(*!
<summary>Checks complete STRING/WSTRING ordering beyond the first 255 characters.</summary>
<description>
Builds equal 260-character prefixes followed by different code units. Exercises both operand directions and
both configuration paths, with properly terminated persistent source storage and owned reference snapshots.
Narrow fixture offsets refer to ASCII bytes, including the explicit terminator at offset 261.
</description>
<param name="assertions">Valid assertion context borrowed from the active case.</param>
*)
METHOD PRIVATE testMixedTextComparison
VAR_INPUT
	assertions : REFERENCE TO TOF_Testing.Assertions;
END_VAR
VAR
	i : INT;
END_VAR
_PairComparisonCondition.Comparer := 0;

// SA0175: Build a 260-byte ASCII prefix, one differing byte and a terminator within persistent storage.
{analysis -175}
FOR i := 0 TO 259 DO
	_ComparisonText[i] := BYTE#16#41;
	_ComparisonWideText[i] := WORD#16#41;
END_FOR

_ComparisonText[260] := BYTE#16#42;
_ComparisonWideText[260] := WORD#16#43;
_ComparisonText[261] := TO_BYTE(TOF_Core.UnsignedInt8.MIN_VALUE);
_ComparisonWideText[261] := TO_WORD(TOF_Core.UnsignedInt16.MIN_VALUE);
{analysis +175}

_PairComparisonCondition.BindPlcVariable(name := 'TextNarrow', plcVariable := _ComparisonText);
_PairComparisonCondition.BindPlcVariable(name := 'TextWide', plcVariable := _ComparisonWideText);

_PairComparisonCondition.ConfigureVariable(
	firstVariableName := 'TextNarrow',
	comparisonOperator := TOF_Workflow.COMPARISON_OPERATOR.LESS_THAN,
	secondVariableName := 'TextWide'
);
assertions.ThatBool(
	actual := _PairComparisonCondition.Evaluate(activity := 0),
	message := "Mixed text must compare beyond character 255"
).IsTrue();

_PairComparisonCondition.ConfigureVariable(
	firstVariableName := 'TextWide',
	comparisonOperator := TOF_Workflow.COMPARISON_OPERATOR.GREATER_THAN,
	secondVariableName := 'TextNarrow'
);
assertions.ThatBool(
	actual := _PairComparisonCondition.Evaluate(activity := 0),
	message := "Reversing mixed encodings must reverse order"
).IsTrue();

_PairComparisonCondition.Configure(
	firstVariableName := 'TextNarrow',
	comparisonOperator := TOF_Workflow.COMPARISON_OPERATOR.LESS_THAN,
	referenceValue := _ComparisonWideText
);
assertions.ThatBool(
	actual := _PairComparisonCondition.Evaluate(activity := 0),
	message := "A long WSTRING reference must compare fully"
).IsTrue();

_PairComparisonCondition.Configure(
	firstVariableName := 'TextWide',
	comparisonOperator := TOF_Workflow.COMPARISON_OPERATOR.GREATER_THAN,
	referenceValue := _ComparisonText
);
assertions.ThatBool(
	actual := _PairComparisonCondition.Evaluate(activity := 0),
	message := "A long STRING reference must compare fully"
).IsTrue();
END_METHOD

(*!
<summary>Checks that equal-category time-of-day and user-defined pairs retain standard comparer dispatch.</summary>
<description>
Uses categories unsupported by built-in GENERIC_VALUE.CompareTo. Time-of-day values retain native order and
user-defined unions retain explicit byte order, including when a reference snapshot is configured.
</description>
<param name="assertions">Valid assertion context borrowed from the active case.</param>
*)
METHOD PRIVATE testStandardComparisonFallback
VAR_INPUT
	assertions : REFERENCE TO TOF_Testing.Assertions;
END_VAR
_PairComparisonCondition.Comparer := 0;
_FirstComparisonBytes.Raw := UDINT#16#01010101;
_SecondComparisonBytes.Raw := UDINT#16#02020202;

_PairComparisonCondition.BindPlcVariable(name := 'FallbackEarlierTime', plcVariable := _FirstComparisonTimeOfDay);
_PairComparisonCondition.BindPlcVariable(name := 'FallbackLaterTime', plcVariable := _SecondComparisonTimeOfDay);
_PairComparisonCondition.BindPlcVariable(name := 'FallbackFirstBytes', plcVariable := _FirstComparisonBytes);
_PairComparisonCondition.BindPlcVariable(name := 'FallbackSecondBytes', plcVariable := _SecondComparisonBytes);

_PairComparisonCondition.ConfigureVariable(
	firstVariableName := 'FallbackEarlierTime',
	comparisonOperator := TOF_Workflow.COMPARISON_OPERATOR.LESS_THAN,
	secondVariableName := 'FallbackLaterTime'
);
assertions.ThatBool(
	actual := _PairComparisonCondition.Evaluate(activity := 0),
	message := "TIME_OF_DAY must retain native ordering"
).IsTrue();

_PairComparisonCondition.Configure(
	firstVariableName := 'FallbackLaterTime',
	comparisonOperator := TOF_Workflow.COMPARISON_OPERATOR.GREATER_THAN,
	referenceValue := _FirstComparisonTimeOfDay
);
assertions.ThatBool(
	actual := _PairComparisonCondition.Evaluate(activity := 0),
	message := "A time-of-day reference must remain supported"
).IsTrue();

_PairComparisonCondition.ConfigureVariable(
	firstVariableName := 'FallbackFirstBytes',
	comparisonOperator := TOF_Workflow.COMPARISON_OPERATOR.LESS_THAN,
	secondVariableName := 'FallbackSecondBytes'
);
assertions.ThatBool(
	actual := _PairComparisonCondition.Evaluate(activity := 0),
	message := "USER_DEFINED must retain byte ordering"
).IsTrue();

_PairComparisonCondition.Configure(
	firstVariableName := 'FallbackSecondBytes',
	comparisonOperator := TOF_Workflow.COMPARISON_OPERATOR.GREATER_THAN,
	referenceValue := _FirstComparisonBytes
);
assertions.ThatBool(
	actual := _PairComparisonCondition.Evaluate(activity := 0),
	message := "A user-defined reference must remain supported"
).IsTrue();
END_METHOD

(*!
<summary>Checks rejection of unrelated categories before standard typed payload comparison.</summary>
<description>
Exercises equal-width numeric/time pairs, numeric/text pairs and OBJECT/USER_DEFINED in both directions.
Both configuration paths are evaluated. Expected exceptions are checked by interface category; a valid
comparison afterwards verifies that failed evaluation preserves reusable configuration state.
</description>
<param name="assertions">Valid assertion context borrowed from the active case.</param>
*)
METHOD PRIVATE testIncompatibleComparisonPairs
VAR_INPUT
	assertions : REFERENCE TO TOF_Testing.Assertions;
END_VAR
_PairComparisonCondition.Comparer := 0;
_PairComparisonCondition.BindPlcVariable(name := 'RejectedNumber', plcVariable := _ComparisonUnrelatedInteger);
_PairComparisonCondition.BindPlcVariable(name := 'RejectedTime', plcVariable := _FirstComparisonTimeOfDay);
_PairComparisonCondition.BindPlcVariable(name := 'RejectedText', plcVariable := _ComparisonText);
_PairComparisonCondition.BindPlcVariable(name := 'RejectedBytes', plcVariable := _FirstComparisonBytes);
_PairComparisonCondition.BindPlcVariable(
	name := 'RejectedObject',
	plcVariable := _ComparisonObject,
	plcVariableIsObject := TRUE
);

_PairComparisonCondition.ConfigureVariable(
	firstVariableName := 'RejectedNumber',
	comparisonOperator := TOF_Workflow.COMPARISON_OPERATOR.EQUAL,
	secondVariableName := 'RejectedTime'
);
assertComparisonRejected(
	assertions := assertions,
	scenario := 'DINT/TOD variables');

_PairComparisonCondition.ConfigureVariable(
	firstVariableName := 'RejectedTime',
	comparisonOperator := TOF_Workflow.COMPARISON_OPERATOR.EQUAL,
	secondVariableName := 'RejectedNumber'
);
assertComparisonRejected(
	assertions := assertions,
	scenario := 'TOD/DINT variables');

_PairComparisonCondition.Configure(
	firstVariableName := 'RejectedNumber',
	comparisonOperator := TOF_Workflow.COMPARISON_OPERATOR.EQUAL,
	referenceValue := _FirstComparisonTimeOfDay
);
assertComparisonRejected(
	assertions := assertions,
	scenario := 'DINT/TOD reference');

_PairComparisonCondition.Configure(
	firstVariableName := 'RejectedTime',
	comparisonOperator := TOF_Workflow.COMPARISON_OPERATOR.EQUAL,
	referenceValue := _ComparisonUnrelatedInteger
);
assertComparisonRejected(
	assertions := assertions,
	scenario := 'TOD/DINT reference');

_PairComparisonCondition.ConfigureVariable(
	firstVariableName := 'RejectedNumber',
	comparisonOperator := TOF_Workflow.COMPARISON_OPERATOR.EQUAL,
	secondVariableName := 'RejectedText'
);
assertComparisonRejected(
	assertions := assertions,
	scenario := 'DINT/STRING variables');

_PairComparisonCondition.ConfigureVariable(
	firstVariableName := 'RejectedText',
	comparisonOperator := TOF_Workflow.COMPARISON_OPERATOR.EQUAL,
	secondVariableName := 'RejectedNumber'
);
assertComparisonRejected(
	assertions := assertions,
	scenario := 'STRING/DINT variables');

_PairComparisonCondition.ConfigureVariable(
	firstVariableName := 'RejectedObject',
	comparisonOperator := TOF_Workflow.COMPARISON_OPERATOR.EQUAL,
	secondVariableName := 'RejectedBytes'
);
assertComparisonRejected(
	assertions := assertions,
	scenario := 'OBJECT/USER_DEFINED variables');

_PairComparisonCondition.ConfigureVariable(
	firstVariableName := 'RejectedBytes',
	comparisonOperator := TOF_Workflow.COMPARISON_OPERATOR.EQUAL,
	secondVariableName := 'RejectedObject'
);
assertComparisonRejected(
	assertions := assertions,
	scenario := 'USER_DEFINED/OBJECT variables');

_PairComparisonCondition.Configure(
	firstVariableName := 'RejectedNumber',
	comparisonOperator := TOF_Workflow.COMPARISON_OPERATOR.EQUAL,
	referenceValue := _ComparisonUnrelatedInteger
);
assertions.ThatBool(
	actual := _PairComparisonCondition.Evaluate(activity := 0),
	message := "The condition must remain usable after rejection"
).IsTrue();
END_METHOD

(*!
<summary>Evaluates the configured pair and asserts the expected unsupported-conversion exception category.</summary>
<description>
Converts an expected configuration failure into a test diagnostic. Unexpected exception categories fail the
assertion. Captured exception interfaces remain borrowed within this call and are not retained after task
cleanup. The persistent condition owns all resources across the exception boundary.
</description>
<param name="scenario">Short label identifying the rejected operand pair in assertion diagnostics.</param>
<param name="assertions">Valid assertion context borrowed from the active case.</param>
*)
METHOD PRIVATE assertComparisonRejected
VAR_INPUT
	assertions : REFERENCE TO TOF_Testing.Assertions;
	scenario : STRING(255);
END_VAR
VAR
	exceptionCode : __SYSTEM.ExceptionCode;
	caughtException : TOF_Core.IException;
	conversionException : TOF_Core.IGenericConversionNotSupportedException;
	caughtExpectedException : BOOL;
END_VAR
__TRY
	_PairComparisonCondition.Evaluate(activity := 0);
__CATCH(exceptionCode)
	caughtException := TOF_Core.ExceptionManager.GetLastException(
		exceptionCode := exceptionCode,
		catchPointNamespaceName := NamespaceName,
		catchPointPOUName := __POUNAME(),
		catchPointPosition := __POSITION()
	);
	caughtExpectedException := __QUERYINTERFACE(caughtException, conversionException);
__ENDTRY

assertions.ThatBool(
	actual := caughtExpectedException,
	message := TO_WSTRING(TOF_Core.Strings.Concat255(scenario, ': expected GenericConversionNotSupportedException'))
).IsTrue();
assertions.ThatBool(
	actual := _PairComparisonCondition.Configured,
	message := TO_WSTRING(TOF_Core.Strings.Concat255(scenario, ': rejected evaluation must preserve configuration'))
).IsTrue();
END_METHOD

(*!
<summary>Runs the packaging and inspection workflow through completion and exception recovery.</summary>
<param name="assertions">Valid assertion context borrowed from the active case.</param>
*)
METHOD PRIVATE testEndToEndComprehensiveScenario
VAR_INPUT
	assertions : REFERENCE TO TOF_Testing.Assertions;
END_VAR
VAR
	cycleIndex : INT;
END_VAR
buildScenarioTree();

_Workflow.SensorFeedPart := FALSE; // will be set TRUE by parallelStep
_Workflow.SensorVacuumOk := TRUE;
_Workflow.SensorInspectionOk := TRUE;

assertions.ThatBool(
	actual := _Workflow.StartingAllowed,
	message := "Workflow must allow starting from PASSIVE_READY"
).IsTrue();
_Workflow.RequestStart();

FOR cycleIndex := 1 TO 200 DO
	_Workflow.Execute();

	IF NOT _Workflow.Busy THEN
		EXIT;
	END_IF
END_FOR

assertions.ThatBool(
	actual := _Workflow.State = TOF_Workflow.WORKFLOW_ELEMENT_STATE.PASSIVE_COMPLETED,
	message := "Workflow must complete with PASSIVE_COMPLETED"
).IsTrue();
assertions.ThatInt(
	actual := _Workflow.ProducedCount,
	message := "ProducedCount must equal 1 after WhileActivity and AssignVariableActivity"
).ToBe(expected := 1);
assertions.ThatBool(
	actual := _Workflow.ErrorHandled,
	message := "ErrorHandled must be TRUE after CatchActivity recovered from Try exception"
).IsTrue();
assertions.ThatBool(
	actual := _ThrowingActivity.ThrowCount > 0,
	message := "ThrowingActivity must have executed and thrown"
).IsTrue();
END_METHOD

(*!
<summary>Checks NotCondition using persistent resource-owning fixtures.</summary>
<description>Fixture allocations remain owned by the suite across unexpected exception propagation.</description>
<param name="assertions">Valid assertion context borrowed from the active case.</param>
*)
METHOD PRIVATE testNotCondition
VAR_INPUT
	assertions : REFERENCE TO TOF_Testing.Assertions;
END_VAR
VAR_INST
	notCond : TOF_Workflow.NotCondition(workflow := _NotWorkflow);
	trueCond : TOF_Workflow.TrueCondition(workflow := _NotWorkflow);
	varCond : TOF_Workflow.VariableHasValueCondition(workflow := _NotWorkflow);
	testVal : INT := 10;
END_VAR
_NotWorkflow.SetRootActivity(rootActivity := _NotRoot);

assertions.ThatBool(
	actual := notCond.Configured,
	message := "NotCondition must not be configured initially"
).IsFalse();

notCond.Configure(condition := trueCond);
assertions.ThatBool(
	actual := notCond.Configured,
	message := "NotCondition must be configured after Configure"
).IsTrue();
assertions.ThatBool(
	actual := notCond.Evaluate(activity := 0),
	message := "NOT True must evaluate to FALSE"
).IsFalse();

_NotWorkflow.ProducedCount := testVal;
varCond.Configure(monitoredVariableName := 'ProducedCount', referenceValue := testVal);
notCond.Configure(condition := varCond);
assertions.ThatBool(
	actual := notCond.Evaluate(activity := 0),
	message := "NOT (ProducedCount = 10) when ProducedCount = 10 must be FALSE"
).IsFalse();

_NotWorkflow.ProducedCount := 99;
assertions.ThatBool(
	actual := notCond.Evaluate(activity := 0),
	message := "NOT (ProducedCount = 10) when ProducedCount = 99 must be TRUE"
).IsTrue();
END_METHOD

(*!
<summary>Checks ParallelActivityWaitAll using persistent resource-owning fixtures.</summary>
<description>Fixture allocations remain owned by the suite across unexpected exception propagation.</description>
<param name="assertions">Valid assertion context borrowed from the active case.</param>
*)
METHOD PRIVATE testParallelActivityWaitAll
VAR_INPUT
	assertions : REFERENCE TO TOF_Testing.Assertions;
END_VAR
VAR_INST
	parallelAct : TOF_Workflow.ParallelActivity(workflow := _WaitAllWorkflow);
	counterTask1 : CounterTask(name := "WaitAllCounter1");
	counterTask2 : CounterTask(name := "WaitAllCounter2");
	taskAct1 : TOF_Workflow.InvokeTaskActivity(workflow := _WaitAllWorkflow);
	taskAct2 : TOF_Workflow.InvokeTaskActivity(workflow := _WaitAllWorkflow);
	cycleIndex : INT;
	refuseReason : TOF_Core.ERROR_MESSAGE;
END_VAR
counterTask1.Reset(refuseReason => refuseReason);
counterTask1.TargetValue := 1;
taskAct1.Configure(task := counterTask1);

counterTask2.Reset(refuseReason => refuseReason);
counterTask2.TargetValue := 2;
taskAct2.Configure(task := counterTask2);

parallelAct.Mode := TOF_Workflow.PARALLEL_JOIN_MODE.WAIT_ALL;
parallelAct.AddChildActivity(activity := taskAct1);
parallelAct.AddChildActivity(activity := taskAct2);

assertions.ThatDInt(actual := parallelAct.ChildCount, message := "ChildCount must be 2").ToBe(expected := 2);

parallelAct.RequestStart();
assertions.ThatBool(
	actual := parallelAct.Busy,
	message := "ParallelActivity must be busy after RequestStart"
).IsTrue();

FOR cycleIndex := 1 TO 50 DO
	parallelAct.Execute();

	IF NOT parallelAct.Busy THEN
		EXIT;
	END_IF
END_FOR

	assertions.ThatBool(
		actual := parallelAct.State = TOF_Workflow.WORKFLOW_ELEMENT_STATE.PASSIVE_COMPLETED,
		message := "ParallelActivity with WAIT_ALL must complete with PASSIVE_COMPLETED"
	).IsTrue();
assertions.ThatBool(
	actual := taskAct1.State = TOF_Workflow.WORKFLOW_ELEMENT_STATE.PASSIVE_COMPLETED,
	message := "taskAct1 must be PASSIVE_COMPLETED"
).IsTrue();
assertions.ThatBool(
	actual := taskAct2.State = TOF_Workflow.WORKFLOW_ELEMENT_STATE.PASSIVE_COMPLETED,
	message := "taskAct2 must be PASSIVE_COMPLETED"
).IsTrue();

parallelAct.RequestReset();
assertions.ThatBool(
	actual := parallelAct.State = TOF_Workflow.WORKFLOW_ELEMENT_STATE.PASSIVE_READY,
	message := "ParallelActivity must reset to PASSIVE_READY"
).IsTrue();
assertions.ThatBool(
	actual := taskAct1.State = TOF_Workflow.WORKFLOW_ELEMENT_STATE.PASSIVE_READY,
	message := "taskAct1 must reset to PASSIVE_READY"
).IsTrue();
assertions.ThatBool(
	actual := taskAct2.State = TOF_Workflow.WORKFLOW_ELEMENT_STATE.PASSIVE_READY,
	message := "taskAct2 must reset to PASSIVE_READY"
).IsTrue();
END_METHOD

(*!
<summary>Checks ParallelActivityWaitAny using persistent resource-owning fixtures.</summary>
<description>Fixture allocations remain owned by the suite across unexpected exception propagation.</description>
<param name="assertions">Valid assertion context borrowed from the active case.</param>
*)
METHOD PRIVATE testParallelActivityWaitAny
VAR_INPUT
	assertions : REFERENCE TO TOF_Testing.Assertions;
END_VAR
VAR_INST
	parallelAct : TOF_Workflow.ParallelActivity(workflow := _WaitAnyWorkflow);
	fastAssign : TOF_Workflow.AssignVariableActivity(workflow := _WaitAnyWorkflow);
	longDelay : TOF_Workflow.DelayActivity(workflow := _WaitAnyWorkflow);
	cycleIndex : INT;
	val : INT := 42;
END_VAR
_WaitAnyWorkflow.SetRootActivity(rootActivity := _WaitAnyRoot);

fastAssign.Configure(targetVariableName := 'ProducedCount', value := val);
longDelay.Interval := T#10S;

parallelAct.Mode := TOF_Workflow.PARALLEL_JOIN_MODE.WAIT_ANY;
parallelAct.AddChildActivity(activity := fastAssign);
parallelAct.AddChildActivity(activity := longDelay);

parallelAct.RequestStart();

FOR cycleIndex := 1 TO 20 DO
	parallelAct.Execute();

	IF NOT parallelAct.Busy THEN
		EXIT;
	END_IF
END_FOR

	assertions.ThatBool(
		actual := parallelAct.State = TOF_Workflow.WORKFLOW_ELEMENT_STATE.PASSIVE_COMPLETED,
		message := "ParallelActivity with WAIT_ANY must complete once fast branch finishes"
	).IsTrue();
assertions.ThatBool(
	actual := fastAssign.State = TOF_Workflow.WORKFLOW_ELEMENT_STATE.PASSIVE_COMPLETED,
	message := "fastAssign must be PASSIVE_COMPLETED"
).IsTrue();
	assertions.ThatBool(
		actual := longDelay.State = TOF_Workflow.WORKFLOW_ELEMENT_STATE.PASSIVE_CANCELLED,
		message := "longDelay must be cancelled when sibling branch completed under WAIT_ANY"
	).IsTrue();

parallelAct.RequestReset();
assertions.ThatBool(
	actual := parallelAct.State = TOF_Workflow.WORKFLOW_ELEMENT_STATE.PASSIVE_READY,
	message := "ParallelActivity must reset to PASSIVE_READY"
).IsTrue();
END_METHOD

(*!
<summary>Checks that a started workflow accepts cancellation and reaches its cancelled state.</summary>
<param name="assertions">Valid assertion context borrowed from the active case.</param>
*)
METHOD PRIVATE testWorkflowCancel
VAR_INPUT
	assertions : REFERENCE TO TOF_Testing.Assertions;
END_VAR
VAR
	cycleIndex : INT;
END_VAR
buildScenarioTree();

_Workflow.SensorVacuumOk := FALSE; // keep waiting at condition
_Workflow.RequestStart();

assertions.ThatBool(
	actual := _Workflow.CancellingAllowed,
	message := "Workflow must allow cancelling while busy"
).IsTrue();
_Workflow.RequestCancel(reason := "Cancelled by test");

FOR cycleIndex := 1 TO 20 DO
	_Workflow.Execute();

	IF NOT _Workflow.Busy THEN
		EXIT;
	END_IF
END_FOR

assertions.ThatBool(
	actual := _Workflow.State = TOF_Workflow.WORKFLOW_ELEMENT_STATE.PASSIVE_CANCELLED,
	message := "Workflow must transition to PASSIVE_CANCELLED"
).IsTrue();
END_METHOD

(*!
<summary>Checks WorkflowReset with an independently prepared workflow fixture.</summary>
<description>
Assertions run unconditionally after preparing the required state; other test outcomes are not prerequisites.
</description>
<param name="assertions">Valid assertion context borrowed from the active case.</param>
*)
METHOD PRIVATE testWorkflowReset
VAR_INPUT
	assertions : REFERENCE TO TOF_Testing.Assertions;
END_VAR
VAR
	cycleIndex : INT;
END_VAR
_ResetActivity.Interval := T#0S;
_ResetWorkflow.SetRootActivity(rootActivity := _ResetActivity);
_ResetWorkflow.ProducedCount := 7;
_ResetWorkflow.ErrorHandled := TRUE;
_ResetWorkflow.RequestStart();

FOR cycleIndex := 1 TO 20 DO
	_ResetWorkflow.Execute();

	IF NOT _ResetWorkflow.Busy THEN
		EXIT;
	END_IF
END_FOR

assertions.ThatBool(
	actual := _ResetWorkflow.State = TOF_Workflow.WORKFLOW_ELEMENT_STATE.PASSIVE_COMPLETED,
	message := "The independent reset fixture must finish its run"
).IsTrue();
assertions.ThatBool(
	actual := _ResetWorkflow.ResettingAllowed,
	message := "A completed workflow must allow reset"
).IsTrue();
_ResetWorkflow.RequestReset();

FOR cycleIndex := 1 TO 20 DO
	_ResetWorkflow.Execute();

	IF NOT _ResetWorkflow.Busy THEN
		EXIT;
	END_IF
END_FOR

assertions.ThatBool(
	actual := _ResetWorkflow.State = TOF_Workflow.WORKFLOW_ELEMENT_STATE.PASSIVE_READY,
	message := "Reset must restore PASSIVE_READY"
).IsTrue();
assertions.ThatInt(
	actual := _ResetWorkflow.ProducedCount,
	message := "Reset must clear ProducedCount"
).ToBe(expected := 0);
assertions.ThatBool(actual := _ResetWorkflow.ErrorHandled, message := "Reset must clear ErrorHandled").IsFalse();
END_METHOD

(*!
<summary>Checks concrete dynamic Workflow creation, variable binding and deletion.</summary>
<description>The suite tracks the pointer persistently until explicit deletion or suite destruction.</description>
<param name="assertions">Valid assertion context borrowed from the active case.</param>
*)
METHOD PRIVATE testDirectWorkflowDynamicCreation
VAR_INPUT
	assertions : REFERENCE TO TOF_Testing.Assertions;
END_VAR
VAR
	resolvedVar : TOF_Core.GENERIC_VALUE;
	registered : BOOL;
	found : BOOL;
END_VAR
_DirectWorkflow := __NEW(TOF_Workflow.Workflow);

IF _DirectWorkflow = 0 THEN
	TOF_Core.DynamicMemoryManager.RaiseAllocationFailure();
END_IF

assertions.ThatBool(
	actual := _DirectWorkflow <> 0,
	message := "Workflow dynamic creation (__NEW) must succeed"
).IsTrue();

IF _DirectWorkflow <> 0 THEN
	registered := _DirectWorkflow^.BindPlcVariable(name := 'DynamicVar', plcVariable := _DynamicTestVar);
	assertions.ThatBool(
		actual := registered,
		message := "BindPlcVariable on dynamic Workflow must return TRUE"
	).IsTrue();

	found := _DirectWorkflow^.TryGetVariable(name := 'DynamicVar', variable => resolvedVar);
	assertions.ThatBool(
		actual := found,
		message := "TryGetVariable on dynamic Workflow must find registered variable"
	).IsTrue();
	assertions.ThatBool(
		actual := resolvedVar.Address = ADR(_DynamicTestVar),
		message := "Resolved variable address must match"
	).IsTrue();

	__DELETE(_DirectWorkflow);
	assertions.ThatBool(
		actual := _DirectWorkflow = 0,
		message := "Workflow dynamic deletion (__DELETE) must succeed"
	).IsTrue();
END_IF
END_METHOD

(*!
<summary>Checks ActivityVariableScopingAndShadowing with an independently prepared workflow fixture.</summary>
<description>
Assertions run unconditionally after preparing the required state; other test outcomes are not prerequisites.
</description>
<param name="assertions">Valid assertion context borrowed from the active case.</param>
*)
METHOD PRIVATE testActivityVariableScopingAndShadowing
VAR_INPUT
	assertions : REFERENCE TO TOF_Testing.Assertions;
END_VAR
VAR
	rootSequence : POINTER TO TOF_Workflow.SequenceActivity;
	childAssign : POINTER TO TOF_Workflow.AssignVariableActivity;
	resolvedVar : TOF_Core.GENERIC_VALUE;
	found : BOOL;
END_VAR
rootSequence := __NEW(TOF_Workflow.SequenceActivity(workflow := _ScopeWorkflow));

IF rootSequence = 0 THEN
	TOF_Core.DynamicMemoryManager.RaiseAllocationFailure();
END_IF

_Workflow.RegisterChild(child := rootSequence^);

childAssign := __NEW(TOF_Workflow.AssignVariableActivity(workflow := _ScopeWorkflow));

IF childAssign = 0 THEN
	TOF_Core.DynamicMemoryManager.RaiseAllocationFailure();
END_IF

_Workflow.RegisterChild(child := childAssign^);

rootSequence^.AddChildActivity(activity := childAssign^);

// Register variable in parent activity scope
rootSequence^.BindPlcVariable(name := 'ParentVar', plcVariable := _ParentScopeVar);

// Child should find parent variable through hierarchical resolution
found := childAssign^.TryGetVariable(name := 'ParentVar', variable => resolvedVar);
assertions.ThatBool(
	actual := found,
	message := "Child activity must resolve variable from parent activity scope"
).IsTrue();
assertions.ThatBool(
	actual := resolvedVar.Address = ADR(_ParentScopeVar),
	message := "Parent variable address must match"
).IsTrue();

// Register variable in workflow, and shadow it in child activity
_ScopeWorkflow.BindPlcVariable(name := 'ShadowVar', plcVariable := _WorkflowScopeVar);
childAssign^.BindPlcVariable(name := 'ShadowVar', plcVariable := _ChildLocalVar);

// Child activity must resolve its own shadowed local variable
found := childAssign^.TryGetVariable(name := 'ShadowVar', variable => resolvedVar);
assertions.ThatBool(actual := found, message := "Child activity must resolve its own shadowed variable").IsTrue();
assertions.ThatBool(
	actual := resolvedVar.Address = ADR(_ChildLocalVar),
	message := "Shadowed variable must point to child local address"
).IsTrue();

// Workflow must resolve its own global variable
found := _ScopeWorkflow.TryGetVariable(name := 'ShadowVar', variable => resolvedVar);
assertions.ThatBool(actual := found, message := "Workflow must resolve its own variable").IsTrue();
assertions.ThatBool(
	actual := resolvedVar.Address = ADR(_WorkflowScopeVar),
	message := "Workflow variable must point to workflow address"
).IsTrue();
END_METHOD

(*!
<summary>Checks VariableRegistrationValidation with an independently prepared workflow fixture.</summary>
<description>
Assertions run unconditionally after preparing the required state; other test outcomes are not prerequisites.
</description>
<param name="assertions">Valid assertion context borrowed from the active case.</param>
*)
METHOD PRIVATE testVariableRegistrationValidation
VAR_INPUT
	assertions : REFERENCE TO TOF_Testing.Assertions;
END_VAR
VAR
	stackValue : INT;
	exceptionCode : __SYSTEM.ExceptionCode;
	exception : TOF_Core.IException;
	configurationException : TOF_Workflow.IWorkflowConfigurationException;
	caughtExpected : BOOL;
END_VAR
_ValidationWorkflow.BindPlcVariable(name := 'Registered', plcVariable := _ValidationValue);

__TRY
	_ValidationWorkflow.BindPlcVariable(name := 'StackValue', plcVariable := stackValue);
__CATCH(exceptionCode)
	exception := TOF_Core.ExceptionManager.GetLastException(
		exceptionCode := exceptionCode,
		catchPointNamespaceName := NamespaceName,
		catchPointPOUName := __POUNAME(),
		catchPointPosition := __POSITION()
	);
	caughtExpected := __QUERYINTERFACE(exception, configurationException);
__ENDTRY

assertions.ThatBool(
	actual := caughtExpected,
	message := "Stack binding must raise WorkflowConfigurationException"
).IsTrue();
caughtExpected := FALSE;

__TRY
	_ValidationWorkflow.BindPlcVariable(name := '', plcVariable := _ValidationValue);
__CATCH(exceptionCode)
	exception := TOF_Core.ExceptionManager.GetLastException(
		exceptionCode := exceptionCode,
		catchPointNamespaceName := NamespaceName,
		catchPointPOUName := __POUNAME(),
		catchPointPosition := __POSITION()
	);
	caughtExpected := __QUERYINTERFACE(exception, configurationException);
__ENDTRY

assertions.ThatBool(
	actual := caughtExpected,
	message := "Empty name must raise WorkflowConfigurationException"
).IsTrue();
caughtExpected := FALSE;

__TRY
	_ValidationWorkflow.BindPlcVariable(name := 'Registered', plcVariable := _ValidationValue);
__CATCH(exceptionCode)
	exception := TOF_Core.ExceptionManager.GetLastException(
		exceptionCode := exceptionCode,
		catchPointNamespaceName := NamespaceName,
		catchPointPOUName := __POUNAME(),
		catchPointPosition := __POSITION()
	);
	caughtExpected := __QUERYINTERFACE(exception, configurationException);
__ENDTRY

assertions.ThatBool(
	actual := caughtExpected,
	message := "Duplicate persistent binding must raise configuration failure"
).IsTrue();

_ValidationActivity.Interval := T#10S;
_ValidationWorkflow.SetRootActivity(rootActivity := _ValidationActivity);
_ValidationWorkflow.RequestStart();
assertions.ThatBool(
	actual := _ValidationWorkflow.Busy,
	message := "The busy guard fixture must actually be active"
).IsTrue();
caughtExpected := FALSE;

__TRY
	_ValidationWorkflow.BindPlcVariable(name := 'WhileBusy', plcVariable := _ValidationValue);
__CATCH(exceptionCode)
	exception := TOF_Core.ExceptionManager.GetLastException(
		exceptionCode := exceptionCode,
		catchPointNamespaceName := NamespaceName,
		catchPointPOUName := __POUNAME(),
		catchPointPosition := __POSITION()
	);
	caughtExpected := __QUERYINTERFACE(exception, configurationException);
__ENDTRY

_ValidationWorkflow.RequestCancel(reason := "Validation complete");
_ValidationWorkflow.RequestReset();
assertions.ThatBool(
	actual := caughtExpected,
	message := "Busy registration must raise configuration failure"
).IsTrue();
END_METHOD

(*!
<summary>Releases any direct-creation fixture still owned by the suite.</summary>
<description>
Completes without exceptions; registered scenario nodes remain owned by their workflow fields.
</description>
*)
METHOD FB_exit : BOOL
VAR_INPUT
	bInCopyCode : BOOL;
END_VAR
IF NOT bInCopyCode AND_THEN _DirectWorkflow <> 0 THEN
	__DELETE(_DirectWorkflow);
END_IF
END_METHOD

END_FUNCTION_BLOCK

// ---- Tests/Workflow/ComprehensiveTestWorkflow.TcPOU
(*
SPDX-FileCopyrightText: © 2026 Oleksandr Tiutyk <trofimich@gmail.com>
SPDX-License-Identifier: MIT
License: https://opensource.org/license/mit
*)

(*!
<summary>Test workflow instance containing named variables for the comprehensive workflow scenario test.</summary>
*)

{attribute 'no_explicit_call' := 'do not call this function block directly'}
{attribute 'enable_dynamic_creation'}
FUNCTION_BLOCK ComprehensiveTestWorkflow EXTENDS TOF_Workflow.Workflow
VAR_INPUT
	SensorFeedPart : BOOL;
	SensorVacuumOk : BOOL;
	SensorInspectionOk : BOOL;
	BatchTarget : INT;
	ProducedCount : INT;
	RejectCount : INT;
	ErrorHandled : BOOL;
END_VAR
VAR_STAT
	//! <summary>Concrete test workflow name available during inherited initialization.</summary>
	_TestWorkflowClassName : STRING := __POUNAME();
END_VAR

METHOD PROTECTED InitializeVariables
BindPlcVariable(name := 'BatchTarget', plcVariable := BatchTarget);
BindPlcVariable(name := 'ProducedCount', plcVariable := ProducedCount);
BindPlcVariable(name := 'RejectCount', plcVariable := RejectCount);
BindPlcVariable(name := 'SensorFeedPart', plcVariable := SensorFeedPart);
BindPlcVariable(name := 'SensorVacuumOk', plcVariable := SensorVacuumOk);
BindPlcVariable(name := 'SensorInspectionOk', plcVariable := SensorInspectionOk);
BindPlcVariable(name := 'ErrorHandled', plcVariable := ErrorHandled);
END_METHOD

{attribute 'monitoring' := 'call'}
PROPERTY NamespaceName : REFERENCE TO STRING
GET
NamespaceName REF= CurrentNamespace.Name;
END_GET
END_PROPERTY

METHOD PROTECTED OnRootActivityRequestReset
VAR_OUTPUT
	abortRequest : BOOL;
END_VAR
ProducedCount := 0;
RejectCount := 0;
ErrorHandled := FALSE;
END_METHOD

{attribute 'monitoring' := 'call'}
PROPERTY SelfSize : ULINT
GET
SelfSize := XSIZEOF(THIS^);
END_GET
END_PROPERTY

(*!
<summary>Returns the concrete test workflow name from initialized static storage.</summary>
*)
{attribute 'monitoring' := 'call'}
PROPERTY ClassName : REFERENCE TO STRING
GET
ClassName REF= _TestWorkflowClassName;
END_GET
END_PROPERTY

END_FUNCTION_BLOCK

// ---- Tests/Workflow/ThrowingTestActivity.TcPOU
(*
SPDX-FileCopyrightText: © 2026 Oleksandr Tiutyk <trofimich@gmail.com>
SPDX-License-Identifier: MIT
License: https://opensource.org/license/mit
*)

(*!
<summary>Test activity that throws a controllable exception during execution for testing TryCatchActivity.</summary>
*)

{attribute 'no_explicit_call' := 'do not call this function block directly'}
{attribute 'enable_dynamic_creation'}
FUNCTION_BLOCK ThrowingTestActivity EXTENDS TOF_Workflow.Activity
VAR_STAT
	{attribute 'hide'}
	_ClassName : STRING := __POUNAME();
END_VAR
VAR
	_ShouldThrow : BOOL := TRUE;
	_ThrowCount : INT;
END_VAR

{attribute 'monitoring' := 'call'}
PROPERTY ClassName : REFERENCE TO STRING
GET
ClassName REF= _ClassName;
END_GET
END_PROPERTY

{attribute 'monitoring' := 'call'}
PROPERTY NamespaceName : REFERENCE TO STRING
GET
NamespaceName REF= CurrentNamespace.Name;
END_GET
END_PROPERTY

METHOD PROTECTED OnResetting : TOF_Workflow.ACTIVITY_RESETTING_STATE
VAR_INPUT
	startResetting : BOOL;
END_VAR
_ThrowCount := 0;
OnResetting := TOF_Workflow.ACTIVITY_RESETTING_STATE.WORK_RESET;
END_METHOD

METHOD PROTECTED OnRunning : TOF_Workflow.ACTIVITY_RUNNING_STATE
VAR_INPUT
	startRunning : BOOL;
	startResuming : BOOL;
END_VAR
VAR_OUTPUT
	haltReason : WSTRING(255);
END_VAR
IF _ShouldThrow THEN
	_ThrowCount := _ThrowCount + 1;
	TOF_Core.Exceptions.ThrowStandard(
		sourceNamespaceName := NamespaceName,
		sourceClassName := ClassName,
		sourcePOUName := __POUNAME(),
		sourcePosition := __POSITION(),
		message := "Controlled exception for TryCatch test"
	);
END_IF

OnRunning := TOF_Workflow.ACTIVITY_RUNNING_STATE.WORK_COMPLETED;
END_METHOD

METHOD PROTECTED OnStopping : TOF_Workflow.ACTIVITY_STOPPING_STATE
VAR_INPUT
	startCancelling : BOOL;
	startSuspending : BOOL;
END_VAR
VAR_OUTPUT
	haltReason : WSTRING(255);
END_VAR
OnStopping := TOF_Workflow.ACTIVITY_STOPPING_STATE.WORK_STOPPED;
END_METHOD

PROPERTY ShouldThrow : BOOL
GET
ShouldThrow := _ShouldThrow;
END_GET
SET
_ShouldThrow := ShouldThrow;
END_SET
END_PROPERTY

PROPERTY ThrowCount : INT
GET
ThrowCount := _ThrowCount;
END_GET
END_PROPERTY

{attribute 'monitoring' := 'call'}
PROPERTY SelfSize : ULINT
GET
SelfSize := XSIZEOF(THIS^);
END_GET
END_PROPERTY

END_FUNCTION_BLOCK

// ---- Tests/Workflow/RecoveryCatchTestActivity.TcPOU
(*
SPDX-FileCopyrightText: © 2026 Oleksandr Tiutyk <trofimich@gmail.com>
SPDX-License-Identifier: MIT
License: https://opensource.org/license/mit
*)

(*!
<summary>Concrete CatchActivity implementation for testing TryCatch exception capture and recovery.</summary>
*)

{attribute 'no_explicit_call' := 'do not call this function block directly'}
{attribute 'enable_dynamic_creation'}
FUNCTION_BLOCK RecoveryCatchTestActivity EXTENDS TOF_Workflow.CatchActivity
VAR_STAT
	{attribute 'hide'}
	_RecoveryCatchClassName : STRING := __POUNAME();
END_VAR
VAR
	_Recovered : BOOL;
END_VAR

//! <summary>Borrows the concrete class name for the lifetime of this instance.</summary>
{attribute 'monitoring' := 'call'}
PROPERTY ClassName : REFERENCE TO STRING
GET
ClassName REF= _RecoveryCatchClassName;
END_GET
END_PROPERTY

{attribute 'monitoring' := 'call'}
PROPERTY NamespaceName : REFERENCE TO STRING
GET
NamespaceName REF= CurrentNamespace.Name;
END_GET
END_PROPERTY

METHOD PROTECTED OnRunning : TOF_Workflow.ACTIVITY_RUNNING_STATE
VAR_INPUT
	startRunning : BOOL;
	startResuming : BOOL;
END_VAR
VAR_OUTPUT
	haltReason : WSTRING(255);
END_VAR
VAR
	variableFound : BOOL;
	errorHandledVar : TOF_Core.GENERIC_VALUE;
	trueValue : BOOL := TRUE;
END_VAR
_Recovered := TRUE;

variableFound := TryGetVariable(name := 'ErrorHandled', variable => errorHandledVar);

IF variableFound THEN
	errorHandledVar.ChangeValueByAnyType(value := trueValue, isObject := FALSE);
END_IF

OnRunning := TOF_Workflow.ACTIVITY_RUNNING_STATE.WORK_COMPLETED;
END_METHOD

METHOD PROTECTED OnStopping : TOF_Workflow.ACTIVITY_STOPPING_STATE
VAR_INPUT
	startCancelling : BOOL;
	startSuspending : BOOL;
END_VAR
VAR_OUTPUT
	haltReason : WSTRING(255);
END_VAR
OnStopping := TOF_Workflow.ACTIVITY_STOPPING_STATE.WORK_STOPPED;
END_METHOD

PROPERTY Recovered : BOOL
GET
Recovered := _Recovered;
END_GET
END_PROPERTY

{attribute 'monitoring' := 'call'}
PROPERTY SelfSize : ULINT
GET
SelfSize := XSIZEOF(THIS^);
END_GET
END_PROPERTY

END_FUNCTION_BLOCK

// ---- Tests/Workflow/WorkflowContractTestGroup.TcPOU
(*
SPDX-FileCopyrightText: © 2026 Oleksandr Tiutyk <trofimich@gmail.com>
SPDX-License-Identifier: MIT
License: https://opensource.org/license/mit
*)

(*!
<summary>Groups workflow ownership, topology, configuration, failure handling and timing scenarios.</summary>
<description>Owns the fixed case tree and runs its leaves in order in the controller task.</description>
*)

{attribute 'no_assign'}
{attribute 'no_explicit_call' := 'do not call this function block directly'}
FUNCTION_BLOCK WorkflowContractTestGroup EXTENDS TOF_Testing.TestGroup<28>
VAR_STAT
	{attribute 'hide'}
	_ClassName : STRING := __POUNAME();
END_VAR
VAR
	_RootAssociation : WorkflowContractTestCase(
		name := "TestRootAssociation",
		parent := THIS^,
		scenario := WORKFLOW_CONTRACT_TEST_SCENARIO.ROOT_ASSOCIATION
	);
	_SequenceTopology : WorkflowContractTestCase(
		name := "TestSequenceTopology",
		parent := THIS^,
		scenario := WORKFLOW_CONTRACT_TEST_SCENARIO.SEQUENCE_TOPOLOGY
	);
	_TransitionDiagnostics : WorkflowContractTestCase(
		name := "TestTransitionDiagnostics",
		parent := THIS^,
		scenario := WORKFLOW_CONTRACT_TEST_SCENARIO.TRANSITION_DIAGNOSTICS
	);
	_DependencyBindings : WorkflowContractTestCase(
		name := "TestDependencyBindings",
		parent := THIS^,
		scenario := WORKFLOW_CONTRACT_TEST_SCENARIO.DEPENDENCY_BINDINGS
	);
	_WriteConfiguration : WorkflowContractTestCase(
		name := "TestWriteConfiguration",
		parent := THIS^,
		scenario := WORKFLOW_CONTRACT_TEST_SCENARIO.WRITE_CONFIGURATION
	);
	_LoadConfiguration : WorkflowContractTestCase(
		name := "TestLoadConfiguration",
		parent := THIS^,
		scenario := WORKFLOW_CONTRACT_TEST_SCENARIO.LOAD_CONFIGURATION
	);
	_OperatorSerialization : WorkflowContractTestCase(
		name := "TestOperatorSerialization",
		parent := THIS^,
		scenario := WORKFLOW_CONTRACT_TEST_SCENARIO.OPERATOR_SERIALIZATION
	);
	_DeserializeNullContextRejection : WorkflowContractTestCase(
		name := "TestDeserializeNullContextRejection",
		parent := THIS^,
		scenario := WORKFLOW_CONTRACT_TEST_SCENARIO.DESERIALIZE_NULL_CONTEXT_REJECTION
	);
	_FactoryDeclarations : WorkflowContractTestCase(
		name := "TestFactoryDeclarations",
		parent := THIS^,
		scenario := WORKFLOW_CONTRACT_TEST_SCENARIO.FACTORY_DECLARATIONS
	);
	_ArrayValidation : WorkflowContractTestCase(
		name := "TestArrayValidation",
		parent := THIS^,
		scenario := WORKFLOW_CONTRACT_TEST_SCENARIO.ARRAY_VALIDATION
	);
	_WorkflowIsolation : WorkflowContractTestCase(
		name := "TestWorkflowIsolation",
		parent := THIS^,
		scenario := WORKFLOW_CONTRACT_TEST_SCENARIO.WORKFLOW_ISOLATION
	);
	_ConditionTopology : WorkflowContractTestCase(
		name := "TestConditionTopology",
		parent := THIS^,
		scenario := WORKFLOW_CONTRACT_TEST_SCENARIO.CONDITION_TOPOLOGY
	);
	_ParentSetters : WorkflowContractTestCase(
		name := "TestParentSetters",
		parent := THIS^,
		scenario := WORKFLOW_CONTRACT_TEST_SCENARIO.PARENT_SETTERS
	);
	_InitializationRetry : WorkflowContractTestCase(
		name := "TestInitializationRetry",
		parent := THIS^,
		scenario := WORKFLOW_CONTRACT_TEST_SCENARIO.INITIALIZATION_RETRY
	);
	_BoundaryDiagnostics : WorkflowContractTestCase(
		name := "TestBoundaryDiagnostics",
		parent := THIS^,
		scenario := WORKFLOW_CONTRACT_TEST_SCENARIO.BOUNDARY_DIAGNOSTICS
	);
	_InvokeConfiguration : WorkflowContractTestCase(
		name := "TestInvokeConfiguration",
		parent := THIS^,
		scenario := WORKFLOW_CONTRACT_TEST_SCENARIO.INVOKE_CONFIGURATION
	);
	_TaskFailureDuringSuspend : WorkflowContractTestCase(
		name := "TestTaskFailureDuringSuspend",
		parent := THIS^,
		scenario := WORKFLOW_CONTRACT_TEST_SCENARIO.TASK_FAILURE_DURING_SUSPEND
	);
	_TaskCompletionDuringSuspend : WorkflowContractTestCase(
		name := "TestTaskCompletionDuringSuspend",
		parent := THIS^,
		scenario := WORKFLOW_CONTRACT_TEST_SCENARIO.TASK_COMPLETION_DURING_SUSPEND
	);
	_TaskAbortDuringSuspend : WorkflowContractTestCase(
		name := "TestTaskAbortDuringSuspend",
		parent := THIS^,
		scenario := WORKFLOW_CONTRACT_TEST_SCENARIO.TASK_ABORT_DURING_SUSPEND
	);
	_TaskReleaseFailureDuringCancel : WorkflowContractTestCase(
		name := "TestTaskReleaseFailureDuringCancel",
		parent := THIS^,
		scenario := WORKFLOW_CONTRACT_TEST_SCENARIO.TASK_RELEASE_FAILURE_DURING_CANCEL
	);
	_CatchCleanupBoundary : WorkflowContractTestCase(
		name := "TestCatchCleanupBoundary",
		parent := THIS^,
		scenario := WORKFLOW_CONTRACT_TEST_SCENARIO.CATCH_CLEANUP_BOUNDARY
	);
	_ConcreteMetadata : WorkflowContractTestCase(
		name := "TestConcreteMetadata",
		parent := THIS^,
		scenario := WORKFLOW_CONTRACT_TEST_SCENARIO.CONCRETE_METADATA
	);
	_VariableLookup : WorkflowContractTestCase(
		name := "TestVariableLookup",
		parent := THIS^,
		scenario := WORKFLOW_CONTRACT_TEST_SCENARIO.VARIABLE_LOOKUP
	);
	_DeclaredVariableReset : WorkflowContractTestCase(
		name := "TestDeclaredVariableReset",
		parent := THIS^,
		scenario := WORKFLOW_CONTRACT_TEST_SCENARIO.DECLARED_VARIABLE_RESET
	);
	_DeclaredVariableValidation : WorkflowContractTestCase(
		name := "TestDeclaredVariableValidation",
		parent := THIS^,
		scenario := WORKFLOW_CONTRACT_TEST_SCENARIO.DECLARED_VARIABLE_VALIDATION
	);
	_ConditionScopePrecedence : WorkflowContractTestCase(
		name := "TestConditionScopePrecedence",
		parent := THIS^,
		scenario := WORKFLOW_CONTRACT_TEST_SCENARIO.CONDITION_SCOPE_PRECEDENCE
	);
	_DelayPauseRemaining : WorkflowDelayPauseRemainingTest(name := "TestDelayPauseRemaining", parent := THIS^);
	_DelayLifecycle : WorkflowContractTestCase(
		name := "TestDelayLifecycle",
		parent := THIS^,
		scenario := WORKFLOW_CONTRACT_TEST_SCENARIO.DELAY_LIFECYCLE
	);
END_VAR
VAR
	_Children : ARRAY [0.._ChildCount - 1] OF TOF_Testing.ITestElement :=
	[
		_RootAssociation,
		_SequenceTopology,
		_TransitionDiagnostics,
		_DependencyBindings,
		_WriteConfiguration,
		_LoadConfiguration,
		_OperatorSerialization,
		_DeserializeNullContextRejection,
		_FactoryDeclarations,
		_ArrayValidation,
		_WorkflowIsolation,
		_ConditionTopology,
		_ParentSetters,
		_InitializationRetry,
		_BoundaryDiagnostics,
		_InvokeConfiguration,
		_TaskFailureDuringSuspend,
		_TaskCompletionDuringSuspend,
		_TaskAbortDuringSuspend,
		_TaskReleaseFailureDuringCancel,
		_CatchCleanupBoundary,
		_ConcreteMetadata,
		_VariableLookup,
		_DeclaredVariableReset,
		_DeclaredVariableValidation,
		_ConditionScopePrecedence,
		_DelayPauseRemaining,
		_DelayLifecycle
	];
END_VAR

(*!
<summary>Borrows the persistent case array. Callers must not modify it.</summary>
*)
{attribute 'monitoring' := 'call'}
PROPERTY Children : REFERENCE TO ARRAY [0.._ChildCount - 1] OF TOF_Testing.ITestElement
GET
Children REF= _Children;
END_GET
END_PROPERTY

(*!
<summary>Borrows the concrete class name. Callers must not modify it.</summary>
*)
{attribute 'monitoring' := 'call'}
PROPERTY ClassName : REFERENCE TO STRING
GET
ClassName REF= _ClassName;
END_GET
END_PROPERTY

(*!
<summary>Borrows the project namespace name. Callers must not modify it.</summary>
*)
{attribute 'monitoring' := 'call'}
PROPERTY NamespaceName : REFERENCE TO STRING
GET
NamespaceName REF= CurrentNamespace.Name;
END_GET
END_PROPERTY

(*!
<summary>Reports the complete instance size in bytes.</summary>
*)
{attribute 'monitoring' := 'call'}
PROPERTY SelfSize : ULINT
GET
SelfSize := XSIZEOF(THIS^);
END_GET
END_PROPERTY

END_FUNCTION_BLOCK

// ---- Tests/Workflow/WorkflowContractTestCase.TcPOU
(*
SPDX-FileCopyrightText: © 2026 Oleksandr Tiutyk <trofimich@gmail.com>
SPDX-License-Identifier: MIT
License: https://opensource.org/license/mit
*)

(*!
<summary>Runs one workflow contract scenario in an isolated fixture.</summary>
<description>
Owns a freshly allocated fixture for the active run. AfterTest releases it after success or a reported
exception. A concrete pointer preserves FB_exit for the fixture and its nested resource owners.
Use one task. Do not copy the test case while it owns a fixture.
</description>
*)

{attribute 'no_assign'}
{attribute 'no_explicit_call' := 'do not call this function block directly'}
FUNCTION_BLOCK WorkflowContractTestCase EXTENDS TOF_Testing.SingleCycleTest
VAR_STAT
	{attribute 'hide'}
	_ClassName : STRING := __POUNAME();
END_VAR
VAR
	_Scenario : WORKFLOW_CONTRACT_TEST_SCENARIO;
	_Fixture : POINTER TO WorkflowContractTestFixture;
END_VAR

(*!
<summary>Selects the scenario without allocating its fixture.</summary>
<param name="name">Name reported for this case.</param>
<param name="parent">Group that owns this case.</param>
<param name="scenario">Scenario selected for the case.</param>
*)
METHOD FB_init : BOOL
VAR_INPUT
	bInitRetains: BOOL; // TRUE: the retain variables are initialized (reset warm / reset cold)
	bInCopyCode: BOOL; // TRUE: the instance will be copied to the copy code afterward (online change)
	name : WSTRING;
	parent : TOF_Testing.ITestElement;
	scenario : WORKFLOW_CONTRACT_TEST_SCENARIO;
END_VAR
IF NOT bInCopyCode THEN
	_Scenario := scenario;
END_IF

FB_init := TRUE;
END_METHOD

(*!
<summary>Allocates a fresh fixture and runs the selected scenario.</summary>
<description>Terminal allocation failure is raised at the task boundary after case handling.</description>
*)
METHOD PROTECTED ExecuteTest
VAR
	assertions : REFERENCE TO TOF_Testing.Assertions;
END_VAR
_Fixture := __NEW(WorkflowContractTestFixture);

IF _Fixture = 0 THEN
	TOF_Core.DynamicMemoryManager.RaiseAllocationFailure();

	RETURN;
END_IF

assertions REF= Assert;
_Fixture^.ExecuteScenario(scenario := _Scenario, assertions := assertions);
END_METHOD

(*!
<summary>Releases the fixture before the case outcome is published.</summary>
<description>The framework records an exception from teardown. Clear the stored alias before releasing.</description>
*)
METHOD PROTECTED AfterTest
VAR
	fixture : POINTER TO WorkflowContractTestFixture;
	released : BOOL;
END_VAR
fixture := _Fixture;
_Fixture := 0;

IF fixture <> 0 THEN
	released := fixture^.TryReleaseLoadedWorkflow();
	__DELETE(fixture);

	IF NOT released THEN
		IF Outcome = TOF_Testing.TEST_OUTCOME.FAILED THEN
			Tc2_System.ADSLOGSTR(
				msgCtrlMask := Tc2_System.Global_Variables.ADSLOG_MSGTYPE_ERROR,
				msgFmtStr := 'Unable to release loaded workflow in %s',
				strArg := TO_STRING(Name)
			);
		ELSE
			RecordFailure(message := "Unable to release loaded workflow");
		END_IF
	END_IF
END_IF
END_METHOD

(*!
<summary>Releases an active fixture if the case is unloaded before its teardown.</summary>
<description>The fixture and its nested FB_exit paths complete without exceptions.</description>
<param name="bInCopyCode">TwinCAT copy-code exit marker. The previous instance leaves copied storage alive.</param>
*)
METHOD FB_exit : BOOL
VAR_INPUT
	bInCopyCode : BOOL;
END_VAR
IF NOT bInCopyCode AND_THEN _Fixture <> 0 THEN
	__DELETE(_Fixture);
END_IF

FB_exit := TRUE;
END_METHOD

(*!
<summary>Borrows the concrete class name. Callers must not modify it.</summary>
*)
{attribute 'monitoring' := 'call'}
PROPERTY ClassName : REFERENCE TO STRING
GET
ClassName REF= _ClassName;
END_GET
END_PROPERTY

(*!
<summary>Borrows the project namespace name. Callers must not modify it.</summary>
*)
{attribute 'monitoring' := 'call'}
PROPERTY NamespaceName : REFERENCE TO STRING
GET
NamespaceName REF= CurrentNamespace.Name;
END_GET
END_PROPERTY

(*!
<summary>Reports the complete instance size in bytes.</summary>
*)
{attribute 'monitoring' := 'call'}
PROPERTY SelfSize : ULINT
GET
SelfSize := XSIZEOF(THIS^);
END_GET
END_PROPERTY

END_FUNCTION_BLOCK

// ---- Tests/Workflow/WorkflowContractTestFixture.TcPOU
(*
SPDX-FileCopyrightText: © 2026 Oleksandr Tiutyk <trofimich@gmail.com>
SPDX-License-Identifier: MIT
License: https://opensource.org/license/mit
*)

(*!
<summary>Owns the state used by one workflow contract test scenario.</summary>
<description>
Each fixture starts with freshly constructed function blocks and stores no borrowed assertion context.
Owns synthetic in-memory workflows and tasks. A dynamically loaded workflow is tracked until checked release.
The case releases it before fixture destruction, including when a scenario reports an exception.
</description>
*)

{attribute 'enable_dynamic_creation'}
{attribute 'no_assign'}
{attribute 'no_explicit_call' := 'do not call this function block directly'}
FUNCTION_BLOCK WorkflowContractTestFixture
	IMPLEMENTS TOF_Workflow.IWorkflowElementFactory,
		TOF_Workflow.IWorkflowDependencyFactory,
		TOF_Workflow.IWorkflowDependencyResolver,
		TOF_Workflow.IWorkflowVariableBinder
VAR_STAT
	//! <summary>Initialized static metadata available during inherited base initialization.</summary>
	_ClassName : STRING := __POUNAME();
END_VAR
VAR
	_LoadSource : TOF_Workflow.Workflow;
	_LoadIf : TOF_Workflow.IfElseActivity(workflow := _LoadSource);
	_LoadCompare : TOF_Workflow.CompareVariableCondition(workflow := _LoadSource);
	_LoadSequence : TOF_Workflow.SequenceActivity(workflow := _LoadSource);
	_LoadEmbeddedInvoke : TOF_Workflow.InvokeTaskActivity(workflow := _LoadSource);
	_LoadExternalInvoke : TOF_Workflow.InvokeTaskActivity(workflow := _LoadSource);
	_LoadAssign : TOF_Workflow.AssignVariableActivity(workflow := _LoadSource);
	_LoadReader : TOF_JSON.JsonConfigurationReader;
	_LoadLoader : TOF_Workflow.WorkflowLoader;
	//! <summary>Owns the loaded workflow until the release check or fixture teardown.</summary>
	_Loaded : TOF_Workflow.IWorkflow;
	_LoadExternal : UINT;
	_BindLoadVariables : BOOL;

	_BindingWorkflow : TOF_Workflow.Workflow;
	_BindingFirst : TOF_Workflow.InvokeTaskActivity(workflow := _BindingWorkflow);
	_BindingSecond : TOF_Workflow.InvokeTaskActivity(workflow := _BindingWorkflow);
	_BindingComparer : TOF_Workflow.CompareVariableCondition(workflow := _BindingWorkflow);
	_BindingExternal : WorkflowBindingTask(name := "External");

	_WriteWorkflow : TOF_Workflow.Workflow;
	_WriteSequence : TOF_Workflow.SequenceActivity(workflow := _WriteWorkflow);
	_WriteDelay : TOF_Workflow.DelayActivity(workflow := _WriteWorkflow);
	_ConfigWriter : TOF_JSON.JsonConfigurationWriter;
	_ConfigDocument : TOF_Core.JSON_DOCUMENT;
	_ConfigParser : Tc3_JsonXml.FB_JsonDomParser;
	_NullContextSequence : TOF_Workflow.SequenceActivity(workflow := 0);
	_NullContextDelay : TOF_Workflow.DelayActivity(workflow := 0);

	_FactoryWorkflow : TOF_Workflow.Workflow;
	_FactoryExits : DINT;
	_ArrayValidation : TOF_Workflow.Workflow;

	_DeclarationWorkflow : TOF_Workflow.Workflow;
	_DeclarationLoop : TOF_Workflow.WhileActivity(workflow := _DeclarationWorkflow);
	_DeclarationGuard : TOF_Workflow.TrueCondition(workflow := _DeclarationWorkflow);
	_DeclarationBody : WorkflowContractActivity(workflow := _DeclarationWorkflow);
	_DeclarationGroup : TOF_Workflow.NotCondition(workflow := _DeclarationWorkflow);
	_DeclarationLeaf : TOF_Workflow.TrueCondition(workflow := _DeclarationWorkflow);
	_DeclarationValidation : TOF_Workflow.Workflow;
	_DeclarationInput : UINT;

	_RootWorkflow : WorkflowContractWorkflow;
	_ForeignWorkflow : TOF_Workflow.Workflow;
	_RootValue : DINT;
	_AssociatedRoot : WorkflowContractActivity(workflow := _RootWorkflow);
	_UnassociatedRoot : WorkflowContractActivity(workflow := 0);
	_ForeignRoot : WorkflowContractActivity(workflow := _ForeignWorkflow);
	_RootPeer : TOF_Workflow.SequenceActivity(workflow := _RootWorkflow);

	_TopologyWorkflow : TOF_Workflow.Workflow;
	_Sequence : TOF_Workflow.SequenceActivity(workflow := _TopologyWorkflow);
	_SequenceFirst : WorkflowContractActivity(workflow := _TopologyWorkflow);
	_SequenceSecond : WorkflowContractActivity(workflow := _TopologyWorkflow);
	_Ancestor : TOF_Workflow.SequenceActivity(workflow := _TopologyWorkflow);
	_Descendant : TOF_Workflow.SequenceActivity(workflow := _TopologyWorkflow);
	_Pick : TOF_Workflow.WaitAndPickActivity(workflow := _TopologyWorkflow);
	_PickFirstCondition : TOF_Workflow.TrueCondition(workflow := _TopologyWorkflow);
	_PickSecondCondition : TOF_Workflow.TrueCondition(workflow := _TopologyWorkflow);
	_PickFirstActivity : WorkflowContractActivity(workflow := _TopologyWorkflow);
	_PickSecondActivity : WorkflowContractActivity(workflow := _TopologyWorkflow);

	_IsolationWorkflow : TOF_Workflow.Workflow;
	_IsolationSequence : TOF_Workflow.SequenceActivity(workflow := _IsolationWorkflow);
	_IsolationParallel : TOF_Workflow.ParallelActivity(workflow := _IsolationWorkflow);
	_IsolationWait : TOF_Workflow.WaitConditionActivity(workflow := _IsolationWorkflow);
	_IsolationWhile : TOF_Workflow.WhileActivity(workflow := _IsolationWorkflow);
	_IsolationIf : TOF_Workflow.IfElseActivity(workflow := _IsolationWorkflow);
	_IsolationNot : TOF_Workflow.NotCondition(workflow := _IsolationWorkflow);
	_IsolationGroup : TOF_Workflow.CompositeCondition(workflow := _IsolationWorkflow);
	_ForeignChild : WorkflowContractActivity(workflow := _ForeignWorkflow);
	_ForeignCondition : TOF_Workflow.TrueCondition(workflow := _ForeignWorkflow);
	_UnassociatedSequence : TOF_Workflow.SequenceActivity(workflow := 0);
	_UnassociatedChild : WorkflowContractActivity(workflow := 0);

	_ConditionWorkflow : TOF_Workflow.Workflow;
	_ConditionGroup : TOF_Workflow.CompositeCondition(workflow := _ConditionWorkflow);
	_ConditionLeaf : TOF_Workflow.TrueCondition(workflow := _ConditionWorkflow);
	_ConditionNot : TOF_Workflow.NotCondition(workflow := _ConditionWorkflow);
	_ConditionHost : TOF_Workflow.WaitConditionActivity(workflow := _ConditionWorkflow);
	_FreeCondition : TOF_Workflow.TrueCondition(workflow := _ConditionWorkflow);

	_ParentWorkflow : TOF_Workflow.Workflow;
	_ParentSequence : TOF_Workflow.SequenceActivity(workflow := _ParentWorkflow);
	_ParentChild : WorkflowContractActivity(workflow := _ParentWorkflow);
	_OtherParent : TOF_Workflow.SequenceActivity(workflow := _ParentWorkflow);
	_ParentCondition : TOF_Workflow.TrueCondition(workflow := _ParentWorkflow);

	_BusyWorkflow : TOF_Workflow.Workflow;
	_BusyRoot : TOF_Workflow.SequenceActivity(workflow := _BusyWorkflow);
	_BusyRunning : WorkflowContractActivity(workflow := _BusyWorkflow);
	_BusyDormant : TOF_Workflow.SequenceActivity(workflow := _BusyWorkflow);
	_BusyCandidate : WorkflowContractActivity(workflow := _BusyWorkflow);

	_RetryWorkflow : WorkflowContractWorkflow;
	_RetryRoot : WorkflowContractActivity(workflow := _RetryWorkflow);
	_ExternalValue : DINT;

	_BoundaryWorkflow : WorkflowContractWorkflow;
	_BoundaryActivity : WorkflowContractActivity(workflow := _BoundaryWorkflow);

	_ConfigWorkflow : TOF_Workflow.Workflow;
	_ConfigActivity : TOF_Workflow.InvokeTaskActivity(workflow := _ConfigWorkflow);
	_ConfigTask : WorkflowContractTask(name := "Configuration task");
	_ReplacementTask : WorkflowContractTask(name := "Replacement task");

	_SuspendFailureWorkflow : TOF_Workflow.Workflow;
	_SuspendFailureActivity : TOF_Workflow.InvokeTaskActivity(workflow := _SuspendFailureWorkflow);
	_SuspendFailureTask : WorkflowContractTask(name := "Suspension failure task");
	_SuspendDoneWorkflow : TOF_Workflow.Workflow;
	_SuspendDoneActivity : TOF_Workflow.InvokeTaskActivity(workflow := _SuspendDoneWorkflow);
	_SuspendDoneTask : WorkflowContractTask(name := "Suspension completion task");
	_SuspendAbortWorkflow : TOF_Workflow.Workflow;
	_SuspendAbortActivity : TOF_Workflow.InvokeTaskActivity(workflow := _SuspendAbortWorkflow);
	_SuspendAbortTask : WorkflowContractTask(name := "Suspension abort task");

	_ReleaseWorkflow : TOF_Workflow.Workflow;
	_ReleaseActivity : TOF_Workflow.InvokeTaskActivity(workflow := _ReleaseWorkflow);
	_ReleaseTask : WorkflowContractTask(name := "Release failure task");
	_ReleaseReplacement : WorkflowContractTask(name := "Release replacement task");
	_ReleaseResource : TaskStoppingResource;

	_CleanupWorkflow : TOF_Workflow.Workflow;
	_CleanupTryCatch : TOF_Workflow.TryCatchActivity(workflow := _CleanupWorkflow);
	_CleanupParallel : TOF_Workflow.ParallelActivity(workflow := _CleanupWorkflow);
	_CleanupInvoke : TOF_Workflow.InvokeTaskActivity(workflow := _CleanupWorkflow);
	_CleanupTask : WorkflowContractTask(name := "Cleanup contract task");
	_CleanupFault : WorkflowContractActivity(workflow := _CleanupWorkflow);
	_CleanupCatch : RecoveryCatchTestActivity(workflow := _CleanupWorkflow);

	_MetadataWorkflow : ComprehensiveTestWorkflow;
	_MetadataBase : TOF_Workflow.Workflow;

	_LookupWorkflow : TOF_Workflow.Workflow;
	_LookupParent : TOF_Workflow.SequenceActivity(workflow := _LookupWorkflow);
	_LookupChild : WorkflowContractActivity(workflow := 0);
	_LookupCondition : TOF_Workflow.TrueCondition(workflow := 0);
	_LookupWorkflowValue : DINT;
	_LookupParentValue : DINT;
	_LookupConditionValue : DINT;

	_ScopeWorkflow : TOF_Workflow.Workflow;
	_ScopeOtherWorkflow : TOF_Workflow.Workflow;
	_ScopeContextParent : TOF_Workflow.SequenceActivity(workflow := _ScopeWorkflow);
	_ScopeContext : WorkflowContractActivity(workflow := _ScopeWorkflow);
	_ScopeAttached : WorkflowContractActivity(workflow := _ScopeWorkflow);
	_ScopeForeignContext : WorkflowContractActivity(workflow := _ScopeOtherWorkflow);
	_ScopeGroup : TOF_Workflow.CompositeCondition(workflow := _ScopeWorkflow);
	_ScopeLeaf : TOF_Workflow.VariableHasValueCondition(workflow := 0);
	_ScopeFree : TOF_Workflow.VariableHasValueCondition(workflow := _ScopeWorkflow);
	_ScopeComparison : TOF_Workflow.CompareVariableCondition(workflow := _ScopeWorkflow);
	_ScopePair : TOF_Workflow.CompareVariableCondition(workflow := _ScopeWorkflow);
	_ScopeLocalValue : DINT := 5;
	_ScopeContextValue : DINT := 20;
	_ScopeAncestorValue : DINT := 30;
	_ScopeConditionParentValue : DINT := 7;
	_ScopeAttachedValue : DINT := 9;
	_ScopeWorkflowValue : DINT := 100;
	_ScopeWorkflowRight : DINT := 101;
	_ScopeOtherValue : DINT := 88;

	_WaitScopeWorkflow : TOF_Workflow.Workflow;
	_WaitScopeActivity : TOF_Workflow.WaitVariableValueActivity(workflow := _WaitScopeWorkflow);

END_VAR

(*!
<summary>Dispatches one scenario against the fresh fixture.</summary>
<description>Call once per fixture. Each method uses the assertions of the receiving case.</description>
<param name="scenario">Scenario assigned to the caller.</param>
<param name="assertions">Valid assertion context borrowed from the active case.</param>
*)
METHOD ExecuteScenario
VAR_INPUT
	scenario : WORKFLOW_CONTRACT_TEST_SCENARIO;
	assertions : REFERENCE TO TOF_Testing.Assertions;
END_VAR
CASE scenario OF
	WORKFLOW_CONTRACT_TEST_SCENARIO.ROOT_ASSOCIATION:
		testRootAssociation(assertions := assertions);

	WORKFLOW_CONTRACT_TEST_SCENARIO.SEQUENCE_TOPOLOGY:
		testSequenceTopology(assertions := assertions);

	WORKFLOW_CONTRACT_TEST_SCENARIO.TRANSITION_DIAGNOSTICS:
		testTransitionDiagnostics(assertions := assertions);

	WORKFLOW_CONTRACT_TEST_SCENARIO.DEPENDENCY_BINDINGS:
		testDependencyBindings(assertions := assertions);

	WORKFLOW_CONTRACT_TEST_SCENARIO.WRITE_CONFIGURATION:
		testWriteConfiguration(assertions := assertions);

	WORKFLOW_CONTRACT_TEST_SCENARIO.LOAD_CONFIGURATION:
		testLoadConfiguration(assertions := assertions);

	WORKFLOW_CONTRACT_TEST_SCENARIO.OPERATOR_SERIALIZATION:
		testOperatorSerialization(assertions := assertions);

	WORKFLOW_CONTRACT_TEST_SCENARIO.DESERIALIZE_NULL_CONTEXT_REJECTION:
		testDeserializeNullContextRejection(assertions := assertions);

	WORKFLOW_CONTRACT_TEST_SCENARIO.FACTORY_DECLARATIONS:
		testFactoryDeclarations(assertions := assertions);

	WORKFLOW_CONTRACT_TEST_SCENARIO.ARRAY_VALIDATION:
		testArrayValidation(assertions := assertions);

	WORKFLOW_CONTRACT_TEST_SCENARIO.WORKFLOW_ISOLATION:
		testWorkflowIsolation(assertions := assertions);

	WORKFLOW_CONTRACT_TEST_SCENARIO.CONDITION_TOPOLOGY:
		testConditionTopology(assertions := assertions);

	WORKFLOW_CONTRACT_TEST_SCENARIO.PARENT_SETTERS:
		testParentSetters(assertions := assertions);

	WORKFLOW_CONTRACT_TEST_SCENARIO.INITIALIZATION_RETRY:
		testInitializationRetry(assertions := assertions);

	WORKFLOW_CONTRACT_TEST_SCENARIO.BOUNDARY_DIAGNOSTICS:
		testBoundaryDiagnostics(assertions := assertions);

	WORKFLOW_CONTRACT_TEST_SCENARIO.INVOKE_CONFIGURATION:
		testInvokeConfiguration(assertions := assertions);

	WORKFLOW_CONTRACT_TEST_SCENARIO.TASK_FAILURE_DURING_SUSPEND:
		testTaskFailureDuringSuspend(assertions := assertions);

	WORKFLOW_CONTRACT_TEST_SCENARIO.TASK_COMPLETION_DURING_SUSPEND:
		testTaskCompletionDuringSuspend(assertions := assertions);

	WORKFLOW_CONTRACT_TEST_SCENARIO.TASK_ABORT_DURING_SUSPEND:
		testTaskAbortDuringSuspend(assertions := assertions);

	WORKFLOW_CONTRACT_TEST_SCENARIO.TASK_RELEASE_FAILURE_DURING_CANCEL:
		testTaskReleaseFailureDuringCancel(assertions := assertions);

	WORKFLOW_CONTRACT_TEST_SCENARIO.CATCH_CLEANUP_BOUNDARY:
		testCatchCleanupBoundary(assertions := assertions);

	WORKFLOW_CONTRACT_TEST_SCENARIO.CONCRETE_METADATA:
		testConcreteMetadata(assertions := assertions);

	WORKFLOW_CONTRACT_TEST_SCENARIO.VARIABLE_LOOKUP:
		testVariableLookup(assertions := assertions);

	WORKFLOW_CONTRACT_TEST_SCENARIO.DECLARED_VARIABLE_RESET:
		testDeclaredVariableReset(assertions := assertions);

	WORKFLOW_CONTRACT_TEST_SCENARIO.DECLARED_VARIABLE_VALIDATION:
		testDeclaredVariableValidation(assertions := assertions);

	WORKFLOW_CONTRACT_TEST_SCENARIO.CONDITION_SCOPE_PRECEDENCE:
		testConditionScopePrecedence(assertions := assertions);

	WORKFLOW_CONTRACT_TEST_SCENARIO.DELAY_LIFECYCLE:
		testDelayLifecycle(assertions := assertions);
ELSE
	assertions.ThatBool(actual := FALSE, message := "Unknown workflow contract scenario").IsTrue();
END_CASE
END_METHOD

(*!
<summary>Borrows the concrete class name. Callers must not modify it.</summary>
*)
{attribute 'monitoring' := 'call'}
PROPERTY ClassName : REFERENCE TO STRING
GET
ClassName REF= _ClassName;
END_GET
END_PROPERTY

(*!
<summary>Borrows the project namespace name. Callers must not modify it.</summary>
*)
{attribute 'monitoring' := 'call'}
PROPERTY NamespaceName : REFERENCE TO STRING
GET
NamespaceName REF= CurrentNamespace.Name;
END_GET
END_PROPERTY

(*!
<summary>Reports the complete instance size in bytes.</summary>
*)
{attribute 'monitoring' := 'call'}
PROPERTY SelfSize : ULINT
GET
SelfSize := XSIZEOF(THIS^);
END_GET
END_PROPERTY

(*!
<summary>Contains a throwing formatter, runs the after-hook once and permits reset and reuse.</summary>
<description>
Uses independently prepared persistent fixtures. Expected failures are checked by exception interface;
ordinary unexpected exceptions leave fixture ownership with the suite.
</description>
<param name="assertions">Valid assertion context borrowed from the active case.</param>
*)
METHOD PRIVATE testBoundaryDiagnostics
VAR_INPUT
	assertions : REFERENCE TO TOF_Testing.Assertions;
END_VAR
VAR
	escaped : BOOL;
END_VAR
_BoundaryWorkflow.SetRootActivity(rootActivity := _BoundaryActivity);
_BoundaryWorkflow.RequestStart();
_BoundaryActivity.throwMessageFailure := TRUE;

__TRY
	_BoundaryWorkflow.Execute();
__CATCH
	escaped := TRUE;
__ENDTRY

assertions.ThatBool(
	actual := escaped,
	message := "Diagnostic conversion must not escape the workflow boundary"
).IsFalse();
assertions.ThatDInt(
	actual := _BoundaryWorkflow.afterCount,
	message := "The after-hook must run once"
).ToBe(expected := 1);
assertions.ThatBool(
	actual := _BoundaryWorkflow.State = TOF_Workflow.WORKFLOW_ELEMENT_STATE.PASSIVE_FAILED,
	message := "The original activity failure must remain visible"
).IsTrue();
assertions.ThatBool(
	actual := _BoundaryWorkflow.FailError.HasError,
	message := "Fallback must be a durable error"
).IsTrue();
assertions.ThatWideString(
	actual := _BoundaryWorkflow.FailError.TopMessage,
	message := "Workflow fallback must identify unavailable diagnostics"
).ToBe(expected := "Workflow exception diagnostics are unavailable");
assertions.ThatWideString(
	actual := _BoundaryActivity.FailError.TopMessage,
	message := "Activity fallback must not retain partial diagnostic output"
).ToBe(expected := "Activity exception diagnostics are unavailable");

assertions.ThatBool(
	actual := _BoundaryWorkflow.FailError.LocalTimestamp = TOF_Core.LongDateAndTimes.EPOCH,
	message := "Fallback must not claim an unavailable exception timestamp"
).IsTrue();
assertions.ThatBool(
	actual := _BoundaryActivity.FailError.LocalTimestamp = TOF_Core.LongDateAndTimes.EPOCH,
	message := "Activity fallback must clear partial timestamps"
).IsTrue();

_BoundaryWorkflow.RequestReset();
assertions.ThatBool(
	actual := _BoundaryWorkflow.FailError.HasError,
	message := "Successful reset must clear fallback diagnostics"
).IsFalse();
_BoundaryActivity.throwMessageFailure := FALSE;
_BoundaryActivity.completeRunning := TRUE;
_BoundaryWorkflow.RequestStart();
assertions.ThatBool(
	actual := _BoundaryWorkflow.State = TOF_Workflow.WORKFLOW_ELEMENT_STATE.PASSIVE_COMPLETED,
	message := "The reset workflow must support a subsequent successful run"
).IsTrue();
END_METHOD

(*!
<summary>Keeps synchronous catch startup separate from pending try-branch cleanup.</summary>
<description>
Uses independent synthetic recovery while a sibling task still stops. Explicit reset must then drive that
remaining work to READY. No physical resource or terminal allocation failure is injected.
</description>
<param name="assertions">Valid assertion context borrowed from the active case.</param>
*)
METHOD PRIVATE testCatchCleanupBoundary
VAR_INPUT
	assertions : REFERENCE TO TOF_Testing.Assertions;
END_VAR
VAR
	i : INT;
END_VAR
_CleanupTask.requiredStopCalls := 3;
_CleanupInvoke.Configure(task := _CleanupTask);
_CleanupFault.throwOrdinaryFailure := TRUE;
_CleanupParallel.AddChildActivity(activity := _CleanupInvoke);
_CleanupParallel.AddChildActivity(activity := _CleanupFault);
_CleanupTryCatch.Configure(tryActivity := _CleanupParallel, catchActivity := _CleanupCatch);
_CleanupWorkflow.SetRootActivity(rootActivity := _CleanupTryCatch);
_CleanupWorkflow.RequestStart();

assertions.ThatBool(
	actual := _CleanupWorkflow.State = TOF_Workflow.WORKFLOW_ELEMENT_STATE.PASSIVE_COMPLETED,
	message := "Independent catch recovery may finish before asynchronous try cleanup"
).IsTrue();
assertions.ThatBool(actual := _CleanupCatch.Recovered, message := "The catch activity must actually run").IsTrue();
assertions.ThatBool(
	actual := _CleanupCatch.Error.HasError,
	message := "Catch diagnostics must be captured synchronously"
).IsTrue();
assertions.ThatBool(
	actual := _CleanupTask.State.Running,
	message := "Failed-branch task cleanup must still be pending"
).IsTrue();
assertions.ThatBool(
	actual := _CleanupWorkflow.Busy,
	message := "Root Busy is not a nested cleanup-completion signal"
).IsFalse();
assertions.ThatDInt(
	actual := _CleanupTask.stopCount,
	message := "Catch startup must not silently drain extra task steps"
).ToBe(expected := 1);

_CleanupWorkflow.RequestReset();

FOR i := 1 TO 8 DO
	_CleanupWorkflow.Execute();

	IF NOT _CleanupWorkflow.Busy THEN
		EXIT;
	END_IF
END_FOR

assertions.ThatBool(
	actual := _CleanupWorkflow.State = TOF_Workflow.WORKFLOW_ELEMENT_STATE.PASSIVE_READY,
	message := "Explicit reset must advance pending try-branch stopping and resetting"
).IsTrue();
assertions.ThatBool(
	actual := _CleanupTask.State.Ready,
	message := "The task must be ready after explicit cleanup"
).IsTrue();
assertions.ThatBool(
	actual := _CleanupCatch.Error.HasError,
	message := "Reset must clear the captured recovery snapshot"
).IsFalse();
END_METHOD

(*!
<summary>Checks concrete workflow metadata without copying ownership-bearing instances.</summary>
<description>
Uses independently prepared persistent fixtures. Expected failures are checked by exception interface;
ordinary unexpected exceptions leave fixture ownership with the suite.
</description>
<param name="assertions">Valid assertion context borrowed from the active case.</param>
*)
METHOD PRIVATE testConcreteMetadata
VAR_INPUT
	assertions : REFERENCE TO TOF_Testing.Assertions;
END_VAR
VAR
	workflowInterface : TOF_Workflow.IWorkflow;
	namedWorkflow : TOF_Core.INamed;
	resetScopeOwner : TOF_Workflow.IVariableResetScopeProvider;
	borrowedResetScope : TOF_Workflow.IVariableResetScope;
END_VAR
assertions.ThatBool(
	actual := _MetadataWorkflow.ClassName = _MetadataBase.ClassName,
	message := "A concrete derived workflow must not report the base workflow class"
).IsFalse();
assertions.ThatString(
	actual := _MetadataWorkflow.NamespaceName,
	message := "The concrete workflow must report the test namespace"
).ToBe(expected := CurrentNamespace.Name);
assertions.ThatULInt(
	actual := _MetadataWorkflow.SelfSize,
	message := "Concrete workflow size must include derived fields"
).ToBe(expected := XSIZEOF(_MetadataWorkflow));
assertions.ThatBool(
	actual := _MetadataWorkflow.SelfAddress = ADR(_MetadataWorkflow),
	message := "Concrete metadata must refer to the original instance"
).IsTrue();

workflowInterface := _MetadataBase;
assertions.ThatBool(
	actual := __QUERYINTERFACE(workflowInterface, namedWorkflow),
	message := "IWorkflow must expose INamed"
).IsTrue();
assertions.ThatBool(
	actual := namedWorkflow.Name <> "",
	message := "Workflow must initialize a default diagnostic name in FB_init"
).IsTrue();
namedWorkflow.Name := "Renamed workflow";
assertions.ThatWideString(
	actual := _MetadataBase.Name,
	message := "Mutating Name through INamed must update the workflow name"
).ToBe(expected := "Renamed workflow");

resetScopeOwner := _AssociatedRoot;
borrowedResetScope := resetScopeOwner.GetResetScope();
assertions.ThatBool(
	actual := borrowedResetScope <> 0,
	message := "Activity must expose its embedded reset scope through IVariableResetScopeProvider"
).IsTrue();

assertions.ThatBool(
	actual := TOF_Workflow.WorkflowExceptions.ClassName <> '',
	message := "The exception helper program must expose its diagnostic name"
).IsTrue();
assertions.ThatBool(
	actual := TOF_Workflow.WorkflowExceptions.ClassName = TOF_Workflow.Workflows.ClassName,
	message := "Different helper programs must retain distinct class metadata"
).IsFalse();
assertions.ThatString(
	actual := TOF_Workflow.WorkflowExceptions.NamespaceName,
	message := "Exception helper namespace must match the workflow library"
).ToBe(expected := _MetadataBase.NamespaceName);
END_METHOD

(*!
<summary>Checks lexical variable precedence in value and relational conditions.</summary>
<description>
Persistent bindings deliberately reuse names with different values. Includes unattached conditions,
condition parents, attached activities, alternate contexts, both comparison operands and workflow fallback.
</description>
<param name="assertions">Valid assertion context borrowed from the active case.</param>
*)
METHOD PRIVATE testConditionScopePrecedence
VAR_INPUT
	assertions : REFERENCE TO TOF_Testing.Assertions;
END_VAR
VAR
	expectedValue : DINT;
	found : BOOL;
	resolved : TOF_Core.GENERIC_VALUE;
END_VAR
_ScopeWorkflow.BindPlcVariable(name := 'Target', plcVariable := _ScopeWorkflowValue);
_ScopeWorkflow.BindPlcVariable(name := 'Right', plcVariable := _ScopeWorkflowRight);
_ScopeWorkflow.BindPlcVariable(name := 'Attached', plcVariable := _ScopeWorkflowValue);
_ScopeWorkflow.BindPlcVariable(name := 'Ancestor', plcVariable := _ScopeWorkflowValue);
_ScopeWorkflow.BindPlcVariable(name := 'WorkflowOnly', plcVariable := _ScopeWorkflowValue);
_ScopeOtherWorkflow.BindPlcVariable(name := 'WorkflowOnly', plcVariable := _ScopeOtherValue);
_ScopeOtherWorkflow.BindPlcVariable(name := 'OtherOnly', plcVariable := _ScopeOtherValue);
_ScopeContext.BindPlcVariable(name := 'Target', plcVariable := _ScopeContextValue);
_ScopeContext.BindPlcVariable(name := 'Right', plcVariable := _ScopeContextValue);
_ScopeContext.BindPlcVariable(name := 'Attached', plcVariable := _ScopeContextValue);
_ScopeContextParent.BindPlcVariable(name := 'Ancestor', plcVariable := _ScopeAncestorValue);
_ScopeContextParent.AddChildActivity(activity := _ScopeContext);

expectedValue := _ScopeContextValue;
_ScopeFree.Configure(monitoredVariableName := 'Target', referenceValue := expectedValue);
assertions.ThatBool(
	actual := _ScopeFree.Evaluate(activity := _ScopeContext),
	message := "Unattached condition must use context local binding before its associated workflow"
).IsTrue();

_ScopeFree.BindPlcVariable(name := 'Target', plcVariable := _ScopeLocalValue);
expectedValue := _ScopeLocalValue;
_ScopeFree.Configure(monitoredVariableName := 'Target', referenceValue := expectedValue);
assertions.ThatBool(
	actual := _ScopeFree.Evaluate(activity := _ScopeContext),
	message := "Condition local binding must shadow context and workflow bindings"
).IsTrue();
assertions.ThatBool(
	actual := _ScopeFree.Evaluate(activity := 0),
	message := "Local binding requires no activity context"
).IsTrue();

_ScopeGroup.BindPlcVariable(name := 'Target', plcVariable := _ScopeConditionParentValue);
_ScopeGroup.AddChildCondition(condition := _ScopeLeaf);
_ScopeGroup.ParentActivity := _ScopeAttached;
_ScopeAttached.BindPlcVariable(name := 'Attached', plcVariable := _ScopeAttachedValue);
expectedValue := _ScopeConditionParentValue;
_ScopeLeaf.Configure(monitoredVariableName := 'Target', referenceValue := expectedValue);
assertions.ThatBool(
	actual := _ScopeLeaf.Evaluate(activity := _ScopeContext),
	message := "Parent condition local binding must precede the evaluating activity"
).IsTrue();

expectedValue := _ScopeAttachedValue;
_ScopeLeaf.Configure(monitoredVariableName := 'Attached', referenceValue := expectedValue);
assertions.ThatBool(
	actual := _ScopeLeaf.Evaluate(activity := _ScopeContext),
	message := "Attached activity binding must precede an alternate evaluating activity"
).IsTrue();

expectedValue := _ScopeAncestorValue;
_ScopeLeaf.Configure(monitoredVariableName := 'Ancestor', referenceValue := expectedValue);
assertions.ThatBool(
	actual := _ScopeLeaf.Evaluate(activity := _ScopeContext),
	message := "Context ancestor binding must precede workflow fallback"
).IsTrue();

expectedValue := _ScopeWorkflowValue;
_ScopeLeaf.Configure(monitoredVariableName := 'WorkflowOnly', referenceValue := expectedValue);
assertions.ThatBool(
	actual := _ScopeLeaf.Evaluate(activity := _ScopeForeignContext),
	message := "Associated workflow fallback must precede a distinct context workflow"
).IsTrue();
assertions.ThatBool(
	actual := _ScopeLeaf.Evaluate(activity := 0),
	message := "Workflow fallback requires no context"
).IsTrue();

expectedValue := _ScopeOtherValue;
_ScopeLeaf.Configure(monitoredVariableName := 'OtherOnly', referenceValue := expectedValue);
assertions.ThatBool(
	actual := _ScopeLeaf.Evaluate(activity := _ScopeForeignContext),
	message := "A distinct context workflow is the last fallback"
).IsTrue();

expectedValue := _ScopeContextValue;
_ScopeComparison.Configure(
	firstVariableName := 'Target',
	comparisonOperator := TOF_Workflow.COMPARISON_OPERATOR.EQUAL,
	referenceValue := expectedValue
);
assertions.ThatBool(
	actual := _ScopeComparison.Evaluate(activity := _ScopeContext),
	message := "Reference comparison must use context locals before workflow fallback"
).IsTrue();
_ScopeComparison.BindPlcVariable(name := 'Target', plcVariable := _ScopeLocalValue);
expectedValue := _ScopeLocalValue;
_ScopeComparison.Configure(
	firstVariableName := 'Target',
	comparisonOperator := TOF_Workflow.COMPARISON_OPERATOR.EQUAL,
	referenceValue := expectedValue
);
assertions.ThatBool(
	actual := _ScopeComparison.Evaluate(activity := _ScopeContext),
	message := "Reference comparison must retain condition-local precedence"
).IsTrue();

_ScopePair.ConfigureVariable(
	firstVariableName := 'Target',
	comparisonOperator := TOF_Workflow.COMPARISON_OPERATOR.EQUAL,
	secondVariableName := 'Right'
);
assertions.ThatBool(
	actual := _ScopePair.Evaluate(activity := _ScopeContext),
	message := "Both comparison operands must resolve in context before workflow fallback"
).IsTrue();

found := _ScopeContext.TryGetLocalVariable(name := 'WorkflowOnly', variable => resolved);
assertions.ThatBool(
	actual := found,
	message := "Local-only activity lookup must not include its workflow"
).IsFalse();
found := _ScopeLeaf.TryGetLocalVariable(name := 'Target', variable => resolved);
assertions.ThatBool(actual := found, message := "Local-only condition lookup must not include its parent").IsFalse();
found := _ScopeFree.TryGetLocalVariable(name := 'Target', variable => resolved);
assertions.ThatBool(actual := found, message := "Direct condition binding must be discoverable").IsTrue();
assertions.ThatBool(
	actual := resolved.Address = ADR(_ScopeLocalValue),
	message := "Local descriptor must remain borrowed"
).IsTrue();

_WaitScopeWorkflow.BindPlcVariable(name := 'Target', plcVariable := _ScopeWorkflowValue);
_WaitScopeActivity.BindPlcVariable(name := 'Target', plcVariable := _ScopeContextValue);
expectedValue := _ScopeContextValue;
_WaitScopeActivity.Configure(monitoredVariableName := 'Target', referenceValue := expectedValue);
_WaitScopeWorkflow.SetRootActivity(rootActivity := _WaitScopeActivity);
_WaitScopeWorkflow.RequestStart();
assertions.ThatBool(
	actual := _WaitScopeWorkflow.State = TOF_Workflow.WORKFLOW_ELEMENT_STATE.PASSIVE_COMPLETED,
	message := "WaitVariableValue internal condition must see the activity local binding before workflow"
).IsTrue();
_WaitScopeWorkflow.RequestReset();
END_METHOD

(*!
<summary>Rejects duplicate and cyclic conditions and resolves activity context through the live chain.</summary>
<description>
Uses independently prepared persistent fixtures. Expected failures are checked by exception interface;
ordinary unexpected exceptions leave fixture ownership with the suite.
</description>
<param name="assertions">Valid assertion context borrowed from the active case.</param>
*)
METHOD PRIVATE testConditionTopology
VAR_INPUT
	assertions : REFERENCE TO TOF_Testing.Assertions;
END_VAR
VAR
	expectedActivity : TOF_Workflow.IActivity;
	expectedCondition : TOF_Workflow.ICondition;
	actualActivity : TOF_Workflow.IActivity;
	actualCondition : TOF_Workflow.ICondition;
	actualElement : TOF_Workflow.IWorkflowElement;
	caught : BOOL;
	exceptionCode : __SYSTEM.ExceptionCode;
	exception : TOF_Core.IException;
	attachmentException : TOF_Workflow.IWorkflowAttachmentException;
END_VAR
_ConditionGroup.AddChildCondition(condition := _ConditionLeaf);
caught := FALSE;

__TRY
	_ConditionGroup.AddChildCondition(condition := _ConditionLeaf);
__CATCH(exceptionCode)
	exception := TOF_Core.ExceptionManager.GetLastException(
		exceptionCode := exceptionCode,
		catchPointNamespaceName := NamespaceName,
		catchPointPOUName := __POUNAME(),
		catchPointPosition := __POSITION()
	);
	caught := __QUERYINTERFACE(exception, attachmentException);
__ENDTRY

assertions.ThatBool(actual := caught, message := "Condition slots cannot share an instance").IsTrue();
_ConditionNot.Configure(condition := _ConditionGroup);
caught := FALSE;

__TRY
	_ConditionGroup.AddChildCondition(condition := _ConditionNot);
__CATCH(exceptionCode)
	exception := TOF_Core.ExceptionManager.GetLastException(
		exceptionCode := exceptionCode,
		catchPointNamespaceName := NamespaceName,
		catchPointPOUName := __POUNAME(),
		catchPointPosition := __POSITION()
	);
	caught := __QUERYINTERFACE(exception, attachmentException);
__ENDTRY

assertions.ThatBool(actual := caught, message := "A condition ancestor cannot become a child").IsTrue();
expectedActivity := _ConditionHost;
_ConditionHost.Configure(condition := _ConditionNot);
_ConditionNot.Configure(condition := _ConditionGroup);
actualActivity := _ConditionLeaf.EnclosingActivity;
assertions.ThatBool(
	actual := actualActivity = expectedActivity,
	message := "Nested condition activity context must follow the parent chain"
).IsTrue();
actualActivity := _ConditionLeaf.ParentActivity;
assertions.ThatBool(
	actual := actualActivity = 0,
	message := "Nested condition immediate parent activity must be zero when attached to a condition"
).IsTrue();
expectedCondition := _ConditionGroup;
actualCondition := _ConditionLeaf.ParentCondition;
assertions.ThatBool(
	actual := actualCondition = expectedCondition,
	message := "Nested condition immediate parent condition must be its direct composite"
).IsTrue();
caught := FALSE;

__TRY
	_ConditionLeaf.ParentCondition := _ConditionLeaf;
__CATCH(exceptionCode)
	exception := TOF_Core.ExceptionManager.GetLastException(
		exceptionCode := exceptionCode,
		catchPointNamespaceName := NamespaceName,
		catchPointPOUName := __POUNAME(),
		catchPointPosition := __POSITION()
	);
	caught := __QUERYINTERFACE(exception, attachmentException);
__ENDTRY

assertions.ThatBool(actual := caught, message := "A bound condition cannot replace its parent").IsTrue();
caught := FALSE;

__TRY
	_FreeCondition.ParentCondition := _FreeCondition;
__CATCH(exceptionCode)
	exception := TOF_Core.ExceptionManager.GetLastException(
		exceptionCode := exceptionCode,
		catchPointNamespaceName := NamespaceName,
		catchPointPOUName := __POUNAME(),
		catchPointPosition := __POSITION()
	);
	caught := __QUERYINTERFACE(exception, attachmentException);
__ENDTRY

assertions.ThatBool(actual := caught, message := "A direct self-parent setter must be rejected").IsTrue();
actualElement := _FreeCondition.Parent;
assertions.ThatBool(
	actual := actualElement = 0,
	message := "Failed setter must preserve an unattached condition"
).IsTrue();
END_METHOD

(*!
<summary>Checks zero interval, same-cycle resume, cancellation and reset reuse.</summary>
<description>
Uses a persistent standalone activity. The positive interval prevents natural completion during synchronous
lifecycle calls; cyclic remaining-time accuracy is covered separately by TestDelayPauseRemaining.
</description>
<param name="assertions">Valid assertion context borrowed from the active case.</param>
*)
METHOD PRIVATE testDelayLifecycle
VAR_INPUT
	assertions : REFERENCE TO TOF_Testing.Assertions;
END_VAR
VAR_INST
	delay : TOF_Workflow.DelayActivity(workflow := 0);
END_VAR
delay.Interval := TOF_Core.Times.MIN_VALUE;
delay.RequestStart();
assertions.ThatBool(
	actual := delay.State = TOF_Workflow.WORKFLOW_ELEMENT_STATE.PASSIVE_COMPLETED,
	message := "Zero interval must complete on a fresh start"
).IsTrue();
delay.RequestReset();
delay.Interval := T#1H;
delay.RequestStart();
delay.RequestSuspend();
delay.RequestStart();
assertions.ThatBool(
	actual := delay.State = TOF_Workflow.WORKFLOW_ELEMENT_STATE.ACTIVE_RUNNING,
	message := "Same-cycle suspension and resume must retain a positive interval"
).IsTrue();
delay.RequestSuspend();
delay.RequestCancel(reason := "Lifecycle regression");
assertions.ThatBool(
	actual := delay.State = TOF_Workflow.WORKFLOW_ELEMENT_STATE.PASSIVE_CANCELLED,
	message := "Cancellation from suspension must finish immediately"
).IsTrue();
assertions.ThatBool(
	actual := delay.Interval = T#1H,
	message := "Cancellation must retain nominal Interval"
).IsTrue();
delay.RequestReset();
delay.RequestStart();
assertions.ThatBool(
	actual := delay.State = TOF_Workflow.WORKFLOW_ELEMENT_STATE.ACTIVE_RUNNING,
	message := "Reset after cancellation must allow another positive run"
).IsTrue();
delay.RequestCancel(reason := "Lifecycle regression cleanup");
delay.RequestReset();
delay.Interval := TOF_Core.Times.MIN_VALUE;
delay.RequestStart();
assertions.ThatBool(
	actual := delay.State = TOF_Workflow.WORKFLOW_ELEMENT_STATE.PASSIVE_COMPLETED,
	message := "Reconfiguring the interval after reset must apply to the next run"
).IsTrue();
delay.RequestReset();
END_METHOD

(*!
<summary>Rolls back only hook-added bindings and retries without deleting caller-owned configuration.</summary>
<description>
Uses independently prepared persistent fixtures. Expected failures are checked by exception interface;
ordinary unexpected exceptions leave fixture ownership with the suite.
</description>
<param name="assertions">Valid assertion context borrowed from the active case.</param>
*)
METHOD PRIVATE testInitializationRetry
VAR_INPUT
	assertions : REFERENCE TO TOF_Testing.Assertions;
END_VAR
VAR
	expectedRoot : TOF_Workflow.IActivity;
	actualActivity : TOF_Workflow.IActivity;
	caught : BOOL;
	exceptionCode : __SYSTEM.ExceptionCode;
	exception : TOF_Core.IException;
	standardException : TOF_Core.IStandardException;
	found : BOOL;
	resolved : TOF_Core.GENERIC_VALUE;
END_VAR
expectedRoot := _RetryRoot;
_RetryWorkflow.BindPlcVariable(name := 'External', plcVariable := _ExternalValue);
_RetryWorkflow.throwInitialization := TRUE;
caught := FALSE;

__TRY
	_RetryWorkflow.SetRootActivity(rootActivity := _RetryRoot);
__CATCH(exceptionCode)
	exception := TOF_Core.ExceptionManager.GetLastException(
		exceptionCode := exceptionCode,
		catchPointNamespaceName := NamespaceName,
		catchPointPOUName := __POUNAME(),
		catchPointPosition := __POSITION()
	);
	caught := __QUERYINTERFACE(exception, standardException);
__ENDTRY

assertions.ThatBool(actual := caught, message := "An ordinary initialization failure must propagate").IsTrue();
actualActivity := _RetryWorkflow.RootActivity;
assertions.ThatBool(
	actual := actualActivity = 0,
	message := "Failed initialization must not install the root"
).IsTrue();
found := _RetryWorkflow.TryGetVariable(name := 'External', variable => resolved);
assertions.ThatBool(
	actual := found,
	message := "A preexisting binding must survive initialization rollback"
).IsTrue();
assertions.ThatBool(
	actual := resolved.Address = ADR(_ExternalValue),
	message := "Preexisting storage identity must survive"
).IsTrue();
found := _RetryWorkflow.TryGetVariable(name := 'Initialized', variable => resolved);
assertions.ThatBool(actual := found, message := "The failed hook binding must be removed").IsFalse();

_RetryWorkflow.SetRootActivity(rootActivity := _RetryRoot);
actualActivity := _RetryWorkflow.RootActivity;
assertions.ThatBool(
	actual := actualActivity = expectedRoot,
	message := "Retry must install the prepared root"
).IsTrue();
assertions.ThatDInt(
	actual := _RetryWorkflow.initializationCount,
	message := "Initialization must retry once"
).ToBe(expected := 2);
found := _RetryWorkflow.TryGetVariable(name := 'Initialized', variable => resolved);
assertions.ThatBool(actual := found, message := "A successful retry must register the hook binding").IsTrue();
_RetryWorkflow.SetRootActivity(rootActivity := _RetryRoot);
assertions.ThatDInt(
	actual := _RetryWorkflow.initializationCount,
	message := "Success must not be initialized again"
).ToBe(expected := 2);
END_METHOD

(*!
<summary>Rejects task replacement while running, stopping and finished, then permits replacement after reset.</summary>
<description>
Uses independently prepared persistent fixtures. Expected failures are checked by exception interface;
ordinary unexpected exceptions leave fixture ownership with the suite.
</description>
<param name="assertions">Valid assertion context borrowed from the active case.</param>
*)
METHOD PRIVATE testInvokeConfiguration
VAR_INPUT
	assertions : REFERENCE TO TOF_Testing.Assertions;
END_VAR
VAR
	expectedTask : TOF_Tasks.ITask;
	actualTask : TOF_Tasks.ITask;
	caught : BOOL;
	exceptionCode : __SYSTEM.ExceptionCode;
	exception : TOF_Core.IException;
	configurationException : TOF_Workflow.IWorkflowConfigurationException;
	i : INT;
END_VAR
expectedTask := _ConfigTask;
_ConfigTask.requiredStopCalls := 3;
_ConfigActivity.Configure(task := _ConfigTask);
_ConfigWorkflow.SetRootActivity(rootActivity := _ConfigActivity);
_ConfigWorkflow.RequestStart();
caught := FALSE;

__TRY
	_ConfigActivity.Configure(task := _ReplacementTask);
__CATCH(exceptionCode)
	exception := TOF_Core.ExceptionManager.GetLastException(
		exceptionCode := exceptionCode,
		catchPointNamespaceName := NamespaceName,
		catchPointPOUName := __POUNAME(),
		catchPointPosition := __POSITION()
	);
	caught := __QUERYINTERFACE(exception, configurationException);
__ENDTRY

assertions.ThatBool(actual := caught, message := "Running configuration must be rejected").IsTrue();
actualTask := _ConfigActivity.Task;
assertions.ThatBool(
	actual := actualTask = expectedTask,
	message := "Rejected replacement preserves the active dependency"
).IsTrue();
_ConfigWorkflow.RequestCancel(reason := "Configuration test");
caught := FALSE;

__TRY
	_ConfigActivity.Configure(task := _ReplacementTask);
__CATCH(exceptionCode)
	exception := TOF_Core.ExceptionManager.GetLastException(
		exceptionCode := exceptionCode,
		catchPointNamespaceName := NamespaceName,
		catchPointPOUName := __POUNAME(),
		catchPointPosition := __POSITION()
	);
	caught := __QUERYINTERFACE(exception, configurationException);
__ENDTRY

assertions.ThatBool(actual := caught, message := "Stopping configuration must be rejected").IsTrue();

FOR i := 1 TO 4 DO
	_ConfigWorkflow.Execute();
END_FOR

assertions.ThatBool(
	actual := _ConfigTask.State.Stopped,
	message := "The original task must be serviced through stopping"
).IsTrue();
caught := FALSE;

__TRY
	_ConfigActivity.Configure(task := _ReplacementTask);
__CATCH(exceptionCode)
	exception := TOF_Core.ExceptionManager.GetLastException(
		exceptionCode := exceptionCode,
		catchPointNamespaceName := NamespaceName,
		catchPointPOUName := __POUNAME(),
		catchPointPosition := __POSITION()
	);
	caught := __QUERYINTERFACE(exception, configurationException);
__ENDTRY

assertions.ThatBool(actual := caught, message := "A finished activity requires reset before configuration").IsTrue();
expectedTask := _ReplacementTask;
_ConfigWorkflow.RequestReset();
_ConfigActivity.Configure(task := _ReplacementTask);
actualTask := _ConfigActivity.Task;
assertions.ThatBool(
	actual := actualTask = expectedTask,
	message := "Ready configuration may replace the dependency"
).IsTrue();
END_METHOD

(*!
<summary>Preserves direct parent links when self, ancestor, detach or replacement assignments are rejected.</summary>
<description>
Uses independently prepared persistent fixtures. Expected failures are checked by exception interface;
ordinary unexpected exceptions leave fixture ownership with the suite.
</description>
<param name="assertions">Valid assertion context borrowed from the active case.</param>
*)
METHOD PRIVATE testParentSetters
VAR_INPUT
	assertions : REFERENCE TO TOF_Testing.Assertions;
END_VAR
VAR
	expectedParent : TOF_Workflow.IActivity;
	actualActivity : TOF_Workflow.IActivity;
	actualElement : TOF_Workflow.IWorkflowElement;
	caught : BOOL;
	exceptionCode : __SYSTEM.ExceptionCode;
	exception : TOF_Core.IException;
	attachmentException : TOF_Workflow.IWorkflowAttachmentException;
	configurationException : TOF_Workflow.IWorkflowConfigurationException;
END_VAR
expectedParent := _ParentSequence;
_ParentSequence.AddChildActivity(activity := _ParentChild);
_ParentChild.ParentActivity := _ParentSequence;
caught := FALSE;

__TRY
	_ParentChild.ParentActivity := _OtherParent;
__CATCH(exceptionCode)
	exception := TOF_Core.ExceptionManager.GetLastException(
		exceptionCode := exceptionCode,
		catchPointNamespaceName := NamespaceName,
		catchPointPOUName := __POUNAME(),
		catchPointPosition := __POSITION()
	);
	caught := __QUERYINTERFACE(exception, attachmentException);
__ENDTRY

assertions.ThatBool(actual := caught, message := "An existing activity parent cannot be replaced").IsTrue();
caught := FALSE;

__TRY
	_ParentChild.ParentActivity := 0;
__CATCH(exceptionCode)
	exception := TOF_Core.ExceptionManager.GetLastException(
		exceptionCode := exceptionCode,
		catchPointNamespaceName := NamespaceName,
		catchPointPOUName := __POUNAME(),
		catchPointPosition := __POSITION()
	);
	caught := __QUERYINTERFACE(exception, attachmentException);
__ENDTRY

assertions.ThatBool(actual := caught, message := "An existing activity parent cannot be detached").IsTrue();
caught := FALSE;

__TRY
	_ParentSequence.ParentActivity := _ParentChild;
__CATCH(exceptionCode)
	exception := TOF_Core.ExceptionManager.GetLastException(
		exceptionCode := exceptionCode,
		catchPointNamespaceName := NamespaceName,
		catchPointPOUName := __POUNAME(),
		catchPointPosition := __POSITION()
	);
	caught := __QUERYINTERFACE(exception, attachmentException);
__ENDTRY

assertions.ThatBool(actual := caught, message := "A direct parent setter cannot create an ancestor cycle").IsTrue();
actualActivity := _ParentChild.ParentActivity;
assertions.ThatBool(
	actual := actualActivity = expectedParent,
	message := "The original parent must be preserved"
).IsTrue();
actualElement := _ParentSequence.Parent;
assertions.ThatBool(actual := actualElement = 0, message := "The ancestor must remain unattached").IsTrue();

_ParentCondition.ParentActivity := _ParentSequence;
caught := FALSE;

__TRY
	_ParentCondition.ParentActivity := _OtherParent;
__CATCH(exceptionCode)
	exception := TOF_Core.ExceptionManager.GetLastException(
		exceptionCode := exceptionCode,
		catchPointNamespaceName := NamespaceName,
		catchPointPOUName := __POUNAME(),
		catchPointPosition := __POSITION()
	);
	caught := __QUERYINTERFACE(exception, attachmentException);
__ENDTRY

assertions.ThatBool(actual := caught, message := "An existing condition parent cannot be replaced").IsTrue();
caught := FALSE;

__TRY
	_ParentCondition.ParentActivity := 0;
__CATCH(exceptionCode)
	exception := TOF_Core.ExceptionManager.GetLastException(
		exceptionCode := exceptionCode,
		catchPointNamespaceName := NamespaceName,
		catchPointPOUName := __POUNAME(),
		catchPointPosition := __POSITION()
	);
	caught := __QUERYINTERFACE(exception, attachmentException);
__ENDTRY

assertions.ThatBool(actual := caught, message := "An existing condition parent cannot be detached").IsTrue();
actualActivity := _ParentCondition.ParentActivity;
assertions.ThatBool(
	actual := actualActivity = expectedParent,
	message := "A condition keeps its original activity parent"
).IsTrue();

_BusyRoot.AddChildActivity(activity := _BusyRunning);
_BusyRoot.AddChildActivity(activity := _BusyDormant);
_BusyWorkflow.SetRootActivity(rootActivity := _BusyRoot);
_BusyWorkflow.RequestStart();
caught := FALSE;

__TRY
	_BusyDormant.AddChildActivity(activity := _BusyCandidate);
__CATCH(exceptionCode)
	exception := TOF_Core.ExceptionManager.GetLastException(
		exceptionCode := exceptionCode,
		catchPointNamespaceName := NamespaceName,
		catchPointPOUName := __POUNAME(),
		catchPointPosition := __POSITION()
	);
	caught := __QUERYINTERFACE(exception, configurationException);
__ENDTRY

assertions.ThatBool(actual := caught, message := "A ready branch in a running tree cannot accept a child").IsTrue();
caught := FALSE;

__TRY
	_BusyCandidate.ParentActivity := _BusyDormant;
__CATCH(exceptionCode)
	exception := TOF_Core.ExceptionManager.GetLastException(
		exceptionCode := exceptionCode,
		catchPointNamespaceName := NamespaceName,
		catchPointPOUName := __POUNAME(),
		catchPointPosition := __POSITION()
	);
	caught := __QUERYINTERFACE(exception, configurationException);
__ENDTRY

assertions.ThatBool(actual := caught, message := "A direct setter cannot mutate a running ancestor tree").IsTrue();
actualElement := _BusyCandidate.Parent;
assertions.ThatBool(
	actual := actualElement = 0,
	message := "Rejected active-tree mutation must preserve the candidate"
).IsTrue();
_BusyWorkflow.RequestCancel(reason := "Topology test complete");
_BusyWorkflow.RequestReset();
END_METHOD

(*!
<summary>Checks explicit root ownership, rejection before mutation and root-child exclusion.</summary>
<description>
Uses independently prepared persistent fixtures. Expected failures are checked by exception interface;
ordinary unexpected exceptions leave fixture ownership with the suite.
</description>
<param name="assertions">Valid assertion context borrowed from the active case.</param>
*)
METHOD PRIVATE testRootAssociation
VAR_INPUT
	assertions : REFERENCE TO TOF_Testing.Assertions;
END_VAR
VAR
	actualActivity : TOF_Workflow.IActivity;
	actualElement : TOF_Workflow.IWorkflowElement;
	caught : BOOL;
	exceptionCode : __SYSTEM.ExceptionCode;
	exception : TOF_Core.IException;
	attachmentException : TOF_Workflow.IWorkflowAttachmentException;
	found : BOOL;
	resolved : TOF_Core.GENERIC_VALUE;
END_VAR
caught := FALSE;

__TRY
	_RootWorkflow.SetRootActivity(rootActivity := _UnassociatedRoot);
__CATCH(exceptionCode)
	exception := TOF_Core.ExceptionManager.GetLastException(
		exceptionCode := exceptionCode,
		catchPointNamespaceName := NamespaceName,
		catchPointPOUName := __POUNAME(),
		catchPointPosition := __POSITION()
	);
	caught := __QUERYINTERFACE(exception, attachmentException);
__ENDTRY

assertions.ThatBool(actual := caught, message := "An unassociated root must be rejected").IsTrue();
actualActivity := _RootWorkflow.RootActivity;
assertions.ThatBool(actual := actualActivity = 0, message := "Rejected root must not be installed").IsTrue();
assertions.ThatDInt(
	actual := _RootWorkflow.initializationCount,
	message := "Validation precedes hooks"
).ToBe(expected := 0);

caught := FALSE;

__TRY
	_RootWorkflow.SetRootActivity(rootActivity := _ForeignRoot);
__CATCH(exceptionCode)
	exception := TOF_Core.ExceptionManager.GetLastException(
		exceptionCode := exceptionCode,
		catchPointNamespaceName := NamespaceName,
		catchPointPOUName := __POUNAME(),
		catchPointPosition := __POSITION()
	);
	caught := __QUERYINTERFACE(exception, attachmentException);
__ENDTRY

assertions.ThatBool(actual := caught, message := "A foreign root must be rejected").IsTrue();

_RootWorkflow.BindPlcVariable(name := 'RootValue', plcVariable := _RootValue);
_RootWorkflow.SetRootActivity(rootActivity := _AssociatedRoot);
_RootWorkflow.SetRootActivity(rootActivity := _AssociatedRoot);
assertions.ThatDInt(
	actual := _RootWorkflow.initializationCount,
	message := "Repeated assignment is a no-op"
).ToBe(expected := 1);
found := _AssociatedRoot.TryGetVariable(name := 'RootValue', variable => resolved);
assertions.ThatBool(actual := found, message := "Associated root must resolve its workflow binding").IsTrue();
assertions.ThatBool(
	actual := resolved.Address = ADR(_RootValue),
	message := "Lookup must retain the borrowed storage"
).IsTrue();

caught := FALSE;

__TRY
	_RootPeer.AddChildActivity(activity := _AssociatedRoot);
__CATCH(exceptionCode)
	exception := TOF_Core.ExceptionManager.GetLastException(
		exceptionCode := exceptionCode,
		catchPointNamespaceName := NamespaceName,
		catchPointPOUName := __POUNAME(),
		catchPointPosition := __POSITION()
	);
	caught := __QUERYINTERFACE(exception, attachmentException);
__ENDTRY

assertions.ThatBool(actual := caught, message := "A registered root must not become a child").IsTrue();
actualElement := _AssociatedRoot.Parent;
assertions.ThatBool(
	actual := actualElement = 0,
	message := "Rejected root attachment must preserve parent"
).IsTrue();
END_METHOD

(*!
<summary>Rejects duplicate, null and cyclic slots and preserves branch-pair ordering after rejection.</summary>
<description>
Uses independently prepared persistent fixtures. Expected failures are checked by exception interface;
ordinary unexpected exceptions leave fixture ownership with the suite.
</description>
<param name="assertions">Valid assertion context borrowed from the active case.</param>
*)
METHOD PRIVATE testSequenceTopology
VAR_INPUT
	assertions : REFERENCE TO TOF_Testing.Assertions;
END_VAR
VAR
	actualElement : TOF_Workflow.IWorkflowElement;
	caught : BOOL;
	exceptionCode : __SYSTEM.ExceptionCode;
	exception : TOF_Core.IException;
	argumentException : TOF_Core.IArgumentNotSpecifiedException;
	attachmentException : TOF_Workflow.IWorkflowAttachmentException;
END_VAR
caught := FALSE;

__TRY
	_Sequence.AddChildActivity(activity := 0);
__CATCH(exceptionCode)
	exception := TOF_Core.ExceptionManager.GetLastException(
		exceptionCode := exceptionCode,
		catchPointNamespaceName := NamespaceName,
		catchPointPOUName := __POUNAME(),
		catchPointPosition := __POSITION()
	);
	caught := __QUERYINTERFACE(exception, argumentException);
__ENDTRY

assertions.ThatBool(actual := caught, message := "Null sequence child must retain its argument exception").IsTrue();
_Sequence.AddChildActivity(activity := _SequenceFirst);
caught := FALSE;

__TRY
	_Sequence.AddChildActivity(activity := _SequenceFirst);
__CATCH(exceptionCode)
	exception := TOF_Core.ExceptionManager.GetLastException(
		exceptionCode := exceptionCode,
		catchPointNamespaceName := NamespaceName,
		catchPointPOUName := __POUNAME(),
		catchPointPosition := __POSITION()
	);
	caught := __QUERYINTERFACE(exception, attachmentException);
__ENDTRY

assertions.ThatBool(actual := caught, message := "An instance may occupy only one sequence slot").IsTrue();
_Sequence.AddChildActivity(activity := _SequenceSecond);

caught := FALSE;

